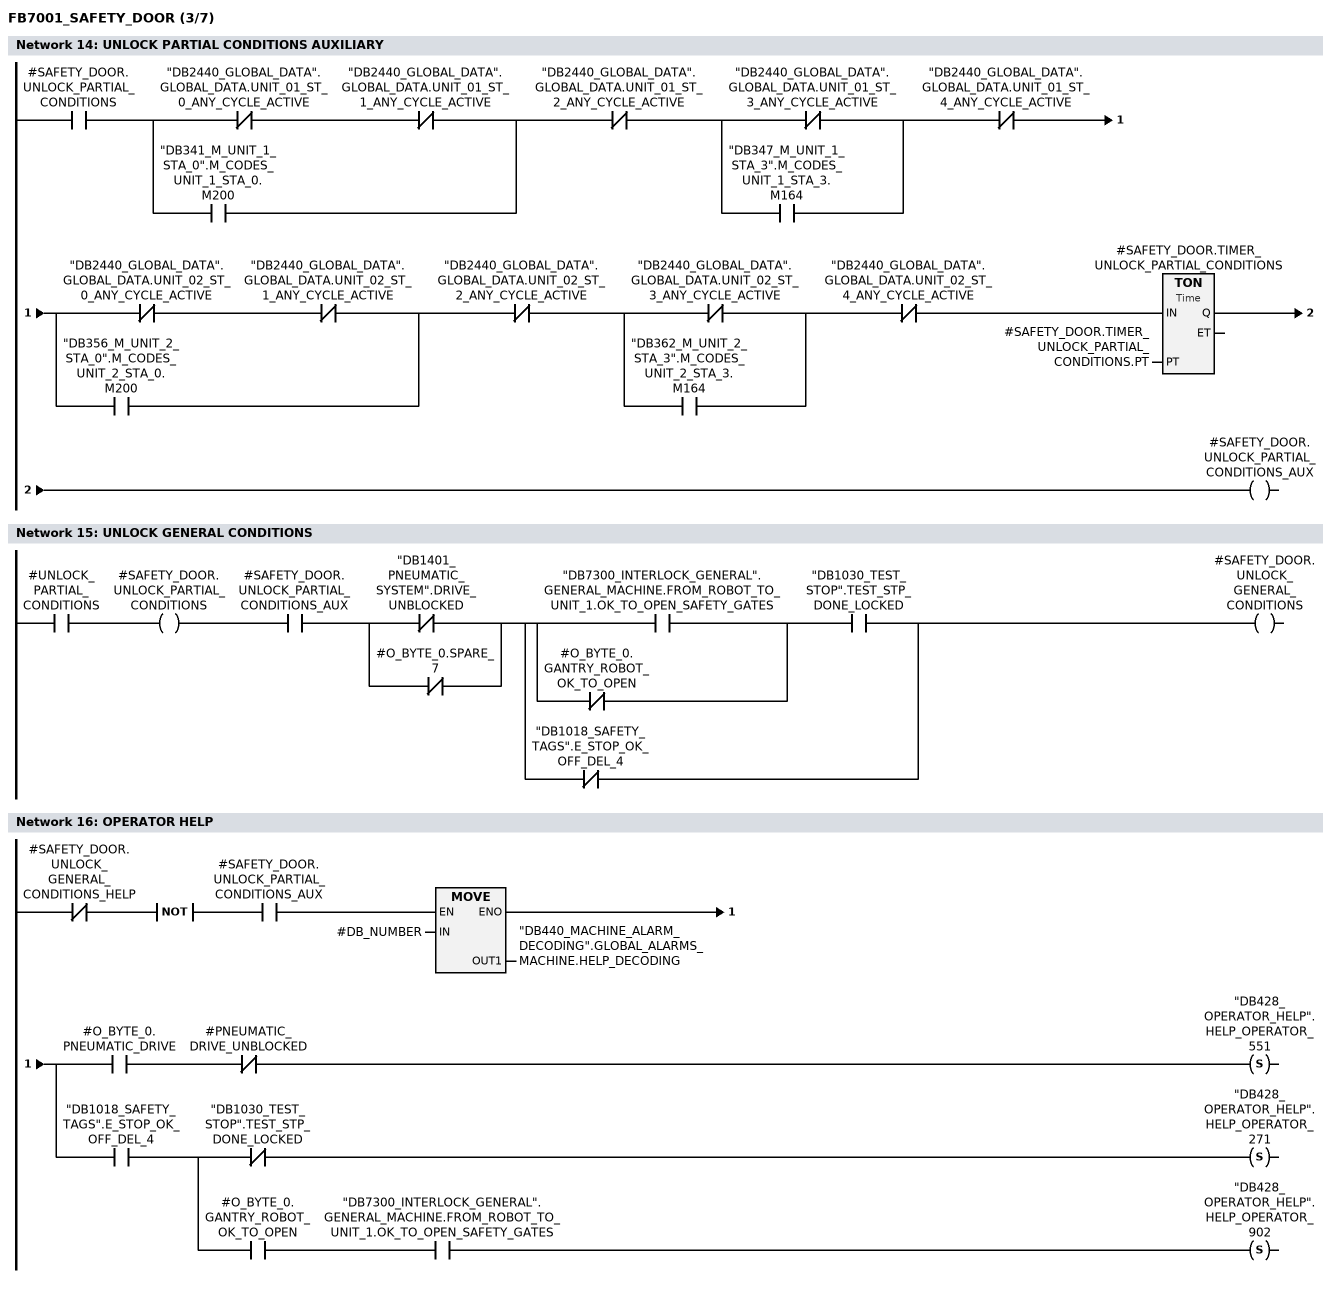
   RUNG wire#powerrail
      Contact( #SAFETY_DOOR.UNLOCK_PARTIAL_CONDITIONS )
      wire#w1
      I_Contact( "DB2440_GLOBAL_DATA".GLOBAL_DATA.UNIT_01_ST_0_ANY_CYCLE_ACTIVE )
      I_Contact( "DB2440_GLOBAL_DATA".GLOBAL_DATA.UNIT_01_ST_1_ANY_CYCLE_ACTIVE )
      wire#w2
      I_Contact( "DB2440_GLOBAL_DATA".GLOBAL_DATA.UNIT_01_ST_2_ANY_CYCLE_ACTIVE )
      wire#w3
      I_Contact( "DB2440_GLOBAL_DATA".GLOBAL_DATA.UNIT_01_ST_3_ANY_CYCLE_ACTIVE )
      wire#w4
      I_Contact( "DB2440_GLOBAL_DATA".GLOBAL_DATA.UNIT_01_ST_4_ANY_CYCLE_ACTIVE )
      wire#w5
      I_Contact( "DB2440_GLOBAL_DATA".GLOBAL_DATA.UNIT_02_ST_0_ANY_CYCLE_ACTIVE )
      I_Contact( "DB2440_GLOBAL_DATA".GLOBAL_DATA.UNIT_02_ST_1_ANY_CYCLE_ACTIVE )
      wire#w6
      I_Contact( "DB2440_GLOBAL_DATA".GLOBAL_DATA.UNIT_02_ST_2_ANY_CYCLE_ACTIVE )
      wire#w7
      I_Contact( "DB2440_GLOBAL_DATA".GLOBAL_DATA.UNIT_02_ST_3_ANY_CYCLE_ACTIVE )
      wire#w8
      I_Contact( "DB2440_GLOBAL_DATA".GLOBAL_DATA.UNIT_02_ST_4_ANY_CYCLE_ACTIVE )
      { S7_Templates := "time_type := Time" } #SAFETY_DOOR.TIMER_UNLOCK_PARTIAL_CONDITIONS.TON(pt := #SAFETY_DOOR.TIMER_UNLOCK_PARTIAL_CONDITIONS.PT, et =>)
      Coil( #SAFETY_DOOR.UNLOCK_PARTIAL_CONDITIONS_AUX )
   END_RUNG
   RUNG wire#w1
      Contact( "DB341_M_UNIT_1_STA_0".M_CODES_UNIT_1_STA_0.M200 )
   END_RUNG wire#w2
   RUNG wire#w3
      Contact( "DB347_M_UNIT_1_STA_3".M_CODES_UNIT_1_STA_3.M164 )
   END_RUNG wire#w4
   RUNG wire#w5
      Contact( "DB356_M_UNIT_2_STA_0".M_CODES_UNIT_2_STA_0.M200 )
   END_RUNG wire#w6
   RUNG wire#w7
      Contact( "DB362_M_UNIT_2_STA_3".M_CODES_UNIT_2_STA_3.M164 )
   END_RUNG wire#w8
   // the same network as SCL:
   #SAFETY_DOOR.TIMER_UNLOCK_PARTIAL_CONDITIONS.TON(IN := #SAFETY_DOOR.UNLOCK_PARTIAL_CONDITIONS AND ((NOT "DB2440_GLOBAL_DATA".GLOBAL_DATA.UNIT_01_ST_0_ANY_CYCLE_ACTIVE AND NOT "DB2440_GLOBAL_DATA".GLOBAL_DATA.UNIT_01_ST_1_ANY_CYCLE_ACTIVE) OR "DB341_M_UNIT_1_STA_0".M_CODES_UNIT_1_STA_0.M200) AND NOT "DB2440_GLOBAL_DATA".GLOBAL_DATA.UNIT_01_ST_2_ANY_CYCLE_ACTIVE AND (NOT "DB2440_GLOBAL_DATA".GLOBAL_DATA.UNIT_01_ST_3_ANY_CYCLE_ACTIVE OR "DB347_M_UNIT_1_STA_3".M_CODES_UNIT_1_STA_3.M164) AND NOT "DB2440_GLOBAL_DATA".GLOBAL_DATA.UNIT_01_ST_4_ANY_CYCLE_ACTIVE AND ((NOT "DB2440_GLOBAL_DATA".GLOBAL_DATA.UNIT_02_ST_0_ANY_CYCLE_ACTIVE AND NOT "DB2440_GLOBAL_DATA".GLOBAL_DATA.UNIT_02_ST_1_ANY_CYCLE_ACTIVE) OR "DB356_M_UNIT_2_STA_0".M_CODES_UNIT_2_STA_0.M200) AND NOT "DB2440_GLOBAL_DATA".GLOBAL_DATA.UNIT_02_ST_2_ANY_CYCLE_ACTIVE AND (NOT "DB2440_GLOBAL_DATA".GLOBAL_DATA.UNIT_02_ST_3_ANY_CYCLE_ACTIVE OR "DB362_M_UNIT_2_STA_3".M_CODES_UNIT_2_STA_3.M164) AND NOT "DB2440_GLOBAL_DATA".GLOBAL_DATA.UNIT_02_ST_4_ANY_CYCLE_ACTIVE,
                           PT := #SAFETY_DOOR.TIMER_UNLOCK_PARTIAL_CONDITIONS.PT);
   #SAFETY_DOOR.UNLOCK_PARTIAL_CONDITIONS_AUX := #SAFETY_DOOR.TIMER_UNLOCK_PARTIAL_CONDITIONS.Q;
END_REGION

REGION Network 15: UNLOCK GENERAL CONDITIONS
   RUNG wire#powerrail
      Contact( #UNLOCK_PARTIAL_CONDITIONS )
      Coil( #SAFETY_DOOR.UNLOCK_PARTIAL_CONDITIONS )
      Contact( #SAFETY_DOOR.UNLOCK_PARTIAL_CONDITIONS_AUX )
      wire#w1
      I_Contact( "DB1401_PNEUMATIC_SYSTEM".DRIVE_UNBLOCKED )
      wire#w2
      Contact( "DB7300_INTERLOCK_GENERAL".GENERAL_MACHINE.FROM_ROBOT_TO_UNIT_1.OK_TO_OPEN_SAFETY_GATES )
      wire#w3
      Contact( "DB1030_TEST_STOP".TEST_STP_DONE_LOCKED )
      wire#w4
      Coil( #SAFETY_DOOR.UNLOCK_GENERAL_CONDITIONS )
   END_RUNG
   RUNG wire#w1
      I_Contact( #O_BYTE_0.SPARE_7 )
   END_RUNG wire#w2
   RUNG wire#w2
      I_Contact( #O_BYTE_0.GANTRY_ROBOT_OK_TO_OPEN )
   END_RUNG wire#w3
   RUNG wire#w2
      I_Contact( "DB1018_SAFETY_TAGS".E_STOP_OK_OFF_DEL_4 )
   END_RUNG wire#w4
   // the same network as SCL:
   #SAFETY_DOOR.UNLOCK_PARTIAL_CONDITIONS := #UNLOCK_PARTIAL_CONDITIONS;
   #SAFETY_DOOR.UNLOCK_GENERAL_CONDITIONS := #UNLOCK_PARTIAL_CONDITIONS AND #SAFETY_DOOR.UNLOCK_PARTIAL_CONDITIONS_AUX AND (NOT "DB1401_PNEUMATIC_SYSTEM".DRIVE_UNBLOCKED OR NOT #O_BYTE_0.SPARE_7) AND ((("DB7300_INTERLOCK_GENERAL".GENERAL_MACHINE.FROM_ROBOT_TO_UNIT_1.OK_TO_OPEN_SAFETY_GATES OR NOT #O_BYTE_0.GANTRY_ROBOT_OK_TO_OPEN) AND "DB1030_TEST_STOP".TEST_STP_DONE_LOCKED) OR NOT "DB1018_SAFETY_TAGS".E_STOP_OK_OFF_DEL_4);
END_REGION

REGION Network 16: OPERATOR HELP
   RUNG wire#powerrail
      I_Contact( #SAFETY_DOOR.UNLOCK_GENERAL_CONDITIONS_HELP )
      Not()
      Contact( #SAFETY_DOOR.UNLOCK_PARTIAL_CONDITIONS_AUX )
      { S7_GenerateENO := "TRUE" } Move(in := #DB_NUMBER, out1 => "DB440_MACHINE_ALARM_DECODING".GLOBAL_ALARMS_MACHINE.HELP_DECODING)
      wire#w1
      Contact( #O_BYTE_0.PNEUMATIC_DRIVE )
      I_Contact( #PNEUMATIC_DRIVE_UNBLOCKED )
      S_Coil( "DB428_OPERATOR_HELP".HELP_OPERATOR_551 )
   END_RUNG
   RUNG wire#w1
      Contact( "DB1018_SAFETY_TAGS".E_STOP_OK_OFF_DEL_4 )
      wire#w2
      I_Contact( "DB1030_TEST_STOP".TEST_STP_DONE_LOCKED )
      S_Coil( "DB428_OPERATOR_HELP".HELP_OPERATOR_271 )
   END_RUNG
   RUNG wire#w2
      Contact( #O_BYTE_0.GANTRY_ROBOT_OK_TO_OPEN )
      Contact( "DB7300_INTERLOCK_GENERAL".GENERAL_MACHINE.FROM_ROBOT_TO_UNIT_1.OK_TO_OPEN_SAFETY_GATES )
      S_Coil( "DB428_OPERATOR_HELP".HELP_OPERATOR_902 )
   END_RUNG
   // the same network as SCL:
   // ENO of a box is taken as its EN; it also drops when the box reports an error
   #_w1 := NOT (NOT #SAFETY_DOOR.UNLOCK_GENERAL_CONDITIONS_HELP) AND #SAFETY_DOOR.UNLOCK_PARTIAL_CONDITIONS_AUX;
   IF #_w1 THEN "DB440_MACHINE_ALARM_DECODING".GLOBAL_ALARMS_MACHINE.HELP_DECODING := #DB_NUMBER; END_IF;
   IF #_w1 AND #O_BYTE_0.PNEUMATIC_DRIVE AND NOT #PNEUMATIC_DRIVE_UNBLOCKED THEN
       "DB428_OPERATOR_HELP".HELP_OPERATOR_551 := TRUE;
   END_IF;
   #_w2 := #_w1 AND "DB1018_SAFETY_TAGS".E_STOP_OK_OFF_DEL_4;
   IF #_w2 AND NOT "DB1030_TEST_STOP".TEST_STP_DONE_LOCKED THEN
       "DB428_OPERATOR_HELP".HELP_OPERATOR_271 := TRUE;
   END_IF;
   IF #_w2 AND #O_BYTE_0.GANTRY_ROBOT_OK_TO_OPEN AND "DB7300_INTERLOCK_GENERAL".GENERAL_MACHINE.FROM_ROBOT_TO_UNIT_1.OK_TO_OPEN_SAFETY_GATES THEN
       "DB428_OPERATOR_HELP".HELP_OPERATOR_902 := TRUE;
   END_IF;
END_REGION

REGION Network 17: UNLOCK MANUAL REQUEST
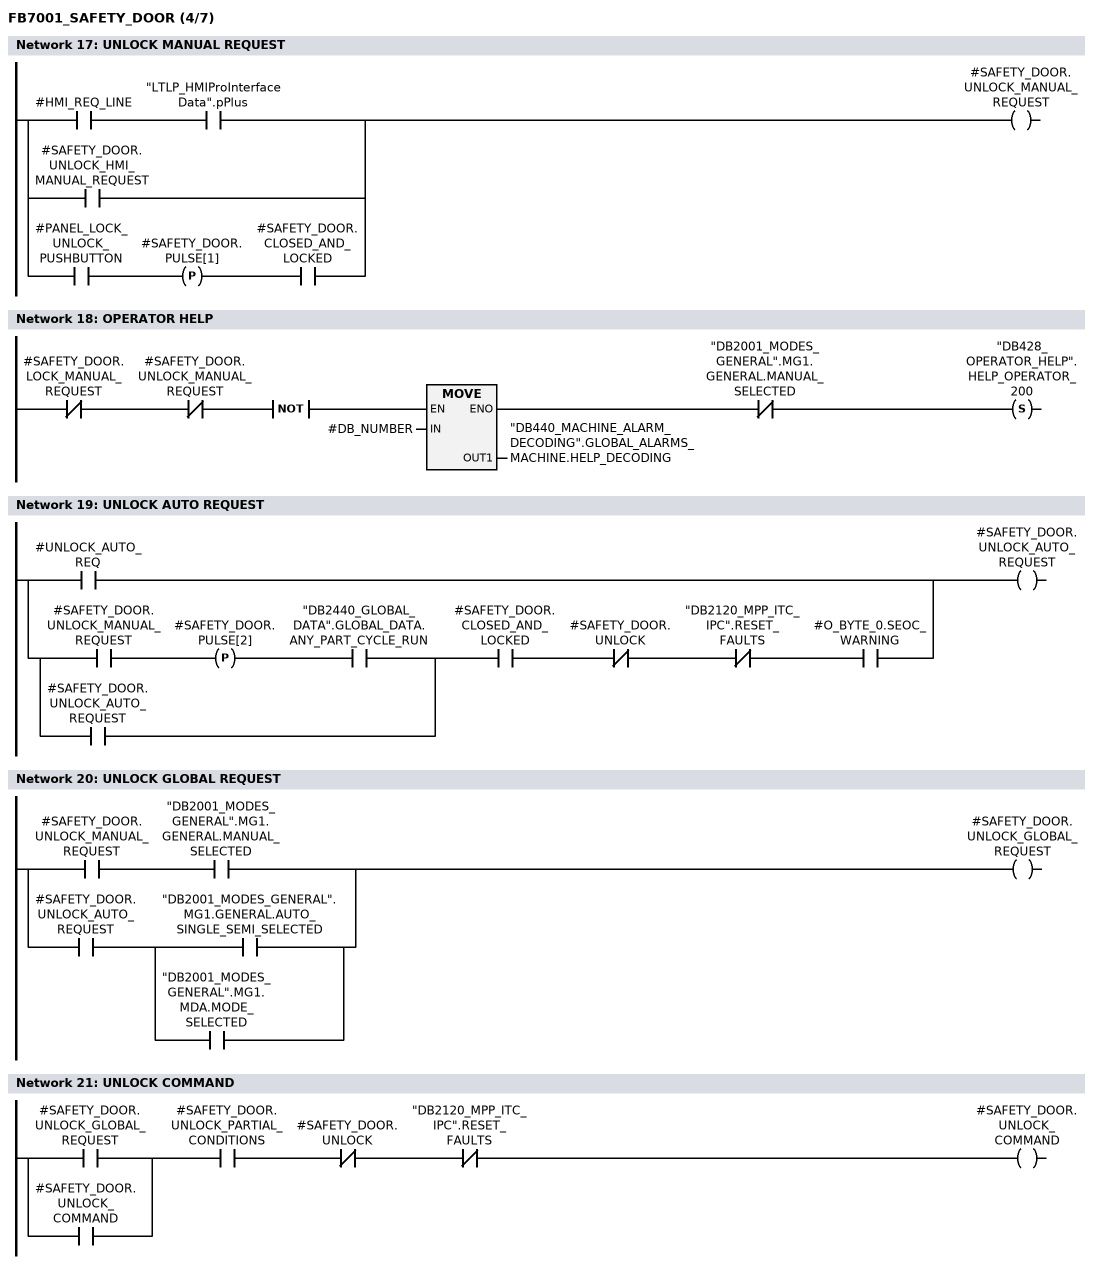
   RUNG wire#powerrail
      Contact( #HMI_REQ_LINE )
      Contact( "LTLP_HMIProInterfaceData".pPlus )
      wire#w1
      Coil( #SAFETY_DOOR.UNLOCK_MANUAL_REQUEST )
   END_RUNG
   RUNG wire#powerrail
      Contact( #SAFETY_DOOR.UNLOCK_HMI_MANUAL_REQUEST )
   END_RUNG wire#w1
   RUNG wire#powerrail
      Contact( #PANEL_LOCK_UNLOCK_PUSHBUTTON )
      P_Trig( #SAFETY_DOOR.PULSE[1] )
      Contact( #SAFETY_DOOR.CLOSED_AND_LOCKED )
   END_RUNG wire#w1
   // the same network as SCL:
   #_w1 := #PANEL_LOCK_UNLOCK_PUSHBUTTON AND NOT #SAFETY_DOOR.PULSE[1];   // rising edge
   #SAFETY_DOOR.PULSE[1] := #PANEL_LOCK_UNLOCK_PUSHBUTTON;
   #SAFETY_DOOR.UNLOCK_MANUAL_REQUEST := (#HMI_REQ_LINE AND "LTLP_HMIProInterfaceData".pPlus) OR #SAFETY_DOOR.UNLOCK_HMI_MANUAL_REQUEST OR (#_w1 AND #SAFETY_DOOR.CLOSED_AND_LOCKED);
END_REGION

REGION Network 18: OPERATOR HELP
   RUNG wire#powerrail
      I_Contact( #SAFETY_DOOR.LOCK_MANUAL_REQUEST )
      I_Contact( #SAFETY_DOOR.UNLOCK_MANUAL_REQUEST )
      Not()
      { S7_GenerateENO := "TRUE" } Move(in := #DB_NUMBER, out1 => "DB440_MACHINE_ALARM_DECODING".GLOBAL_ALARMS_MACHINE.HELP_DECODING)
      I_Contact( "DB2001_MODES_GENERAL".MG1.GENERAL.MANUAL_SELECTED )
      S_Coil( "DB428_OPERATOR_HELP".HELP_OPERATOR_200 )
   END_RUNG
   // the same network as SCL:
   // ENO of a box is taken as its EN; it also drops when the box reports an error
   #_w1 := NOT (NOT #SAFETY_DOOR.LOCK_MANUAL_REQUEST AND NOT #SAFETY_DOOR.UNLOCK_MANUAL_REQUEST);
   IF #_w1 THEN "DB440_MACHINE_ALARM_DECODING".GLOBAL_ALARMS_MACHINE.HELP_DECODING := #DB_NUMBER; END_IF;
   IF #_w1 AND NOT "DB2001_MODES_GENERAL".MG1.GENERAL.MANUAL_SELECTED THEN
       "DB428_OPERATOR_HELP".HELP_OPERATOR_200 := TRUE;
   END_IF;
END_REGION

REGION Network 19: UNLOCK AUTO REQUEST
   RUNG wire#powerrail
      Contact( #UNLOCK_AUTO_REQ )
      wire#w1
      Coil( #SAFETY_DOOR.UNLOCK_AUTO_REQUEST )
   END_RUNG
   RUNG wire#powerrail
      Contact( #SAFETY_DOOR.UNLOCK_MANUAL_REQUEST )
      P_Trig( #SAFETY_DOOR.PULSE[2] )
      Contact( "DB2440_GLOBAL_DATA".GLOBAL_DATA.ANY_PART_CYCLE_RUN )
      wire#w2
      Contact( #SAFETY_DOOR.CLOSED_AND_LOCKED )
      I_Contact( #SAFETY_DOOR.UNLOCK )
      I_Contact( "DB2120_MPP_ITC_IPC".RESET_FAULTS )
      Contact( #O_BYTE_0.SEOC_WARNING )
   END_RUNG wire#w1
   RUNG wire#powerrail
      Contact( #SAFETY_DOOR.UNLOCK_AUTO_REQUEST )
   END_RUNG wire#w2
   // the same network as SCL:
   #_w1 := #SAFETY_DOOR.UNLOCK_MANUAL_REQUEST AND NOT #SAFETY_DOOR.PULSE[2];   // rising edge
   #SAFETY_DOOR.PULSE[2] := #SAFETY_DOOR.UNLOCK_MANUAL_REQUEST;
   #SAFETY_DOOR.UNLOCK_AUTO_REQUEST := #UNLOCK_AUTO_REQ OR (((#_w1 AND "DB2440_GLOBAL_DATA".GLOBAL_DATA.ANY_PART_CYCLE_RUN) OR #SAFETY_DOOR.UNLOCK_AUTO_REQUEST) AND #SAFETY_DOOR.CLOSED_AND_LOCKED AND NOT #SAFETY_DOOR.UNLOCK AND NOT "DB2120_MPP_ITC_IPC".RESET_FAULTS AND #O_BYTE_0.SEOC_WARNING);
END_REGION

REGION Network 20: UNLOCK GLOBAL REQUEST
   RUNG wire#powerrail
      Contact( #SAFETY_DOOR.UNLOCK_MANUAL_REQUEST )
      Contact( "DB2001_MODES_GENERAL".MG1.GENERAL.MANUAL_SELECTED )
      wire#w1
      Coil( #SAFETY_DOOR.UNLOCK_GLOBAL_REQUEST )
   END_RUNG
   RUNG wire#powerrail
      Contact( #SAFETY_DOOR.UNLOCK_AUTO_REQUEST )
      wire#w2
      Contact( "DB2001_MODES_GENERAL".MG1.GENERAL.AUTO_SINGLE_SEMI_SELECTED )
   END_RUNG wire#w1
   RUNG wire#w2
      Contact( "DB2001_MODES_GENERAL".MG1.MDA.MODE_SELECTED )
   END_RUNG wire#w1
   // the same network as SCL:
   #SAFETY_DOOR.UNLOCK_GLOBAL_REQUEST := (#SAFETY_DOOR.UNLOCK_MANUAL_REQUEST AND "DB2001_MODES_GENERAL".MG1.GENERAL.MANUAL_SELECTED) OR (#SAFETY_DOOR.UNLOCK_AUTO_REQUEST AND ("DB2001_MODES_GENERAL".MG1.GENERAL.AUTO_SINGLE_SEMI_SELECTED OR "DB2001_MODES_GENERAL".MG1.MDA.MODE_SELECTED));
END_REGION

REGION Network 21: UNLOCK COMMAND
   RUNG wire#powerrail
      Contact( #SAFETY_DOOR.UNLOCK_GLOBAL_REQUEST )
      wire#w1
      Contact( #SAFETY_DOOR.UNLOCK_PARTIAL_CONDITIONS )
      I_Contact( #SAFETY_DOOR.UNLOCK )
      I_Contact( "DB2120_MPP_ITC_IPC".RESET_FAULTS )
      Coil( #SAFETY_DOOR.UNLOCK_COMMAND )
   END_RUNG
   RUNG wire#powerrail
      Contact( #SAFETY_DOOR.UNLOCK_COMMAND )
   END_RUNG wire#w1
   // the same network as SCL:
   #SAFETY_DOOR.UNLOCK_COMMAND := (#SAFETY_DOOR.UNLOCK_GLOBAL_REQUEST OR #SAFETY_DOOR.UNLOCK_COMMAND) AND #SAFETY_DOOR.UNLOCK_PARTIAL_CONDITIONS AND NOT #SAFETY_DOOR.UNLOCK AND NOT "DB2120_MPP_ITC_IPC".RESET_FAULTS;
END_REGION

REGION Network 22: UNLOCK
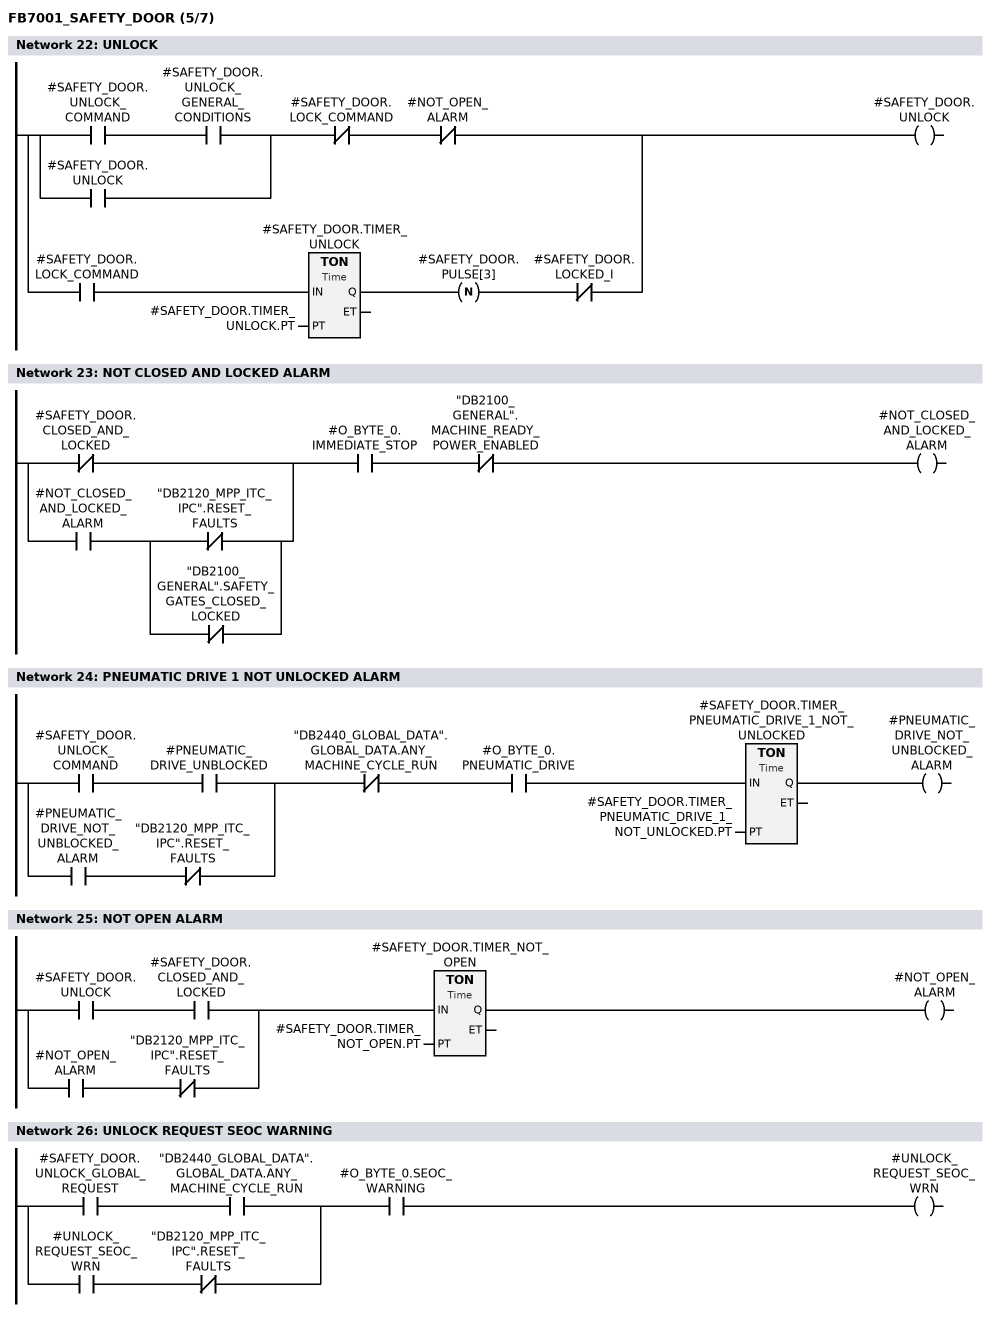
   RUNG wire#powerrail
      Contact( #SAFETY_DOOR.UNLOCK_COMMAND )
      Contact( #SAFETY_DOOR.UNLOCK_GENERAL_CONDITIONS )
      wire#w1
      I_Contact( #SAFETY_DOOR.LOCK_COMMAND )
      I_Contact( #NOT_OPEN_ALARM )
      wire#w2
      Coil( #SAFETY_DOOR.UNLOCK )
   END_RUNG
   RUNG wire#powerrail
      Contact( #SAFETY_DOOR.UNLOCK )
   END_RUNG wire#w1
   RUNG wire#powerrail
      Contact( #SAFETY_DOOR.LOCK_COMMAND )
      { S7_Templates := "time_type := Time" } #SAFETY_DOOR.TIMER_UNLOCK.TON(pt := #SAFETY_DOOR.TIMER_UNLOCK.PT, et =>)
      N_Trig( #SAFETY_DOOR.PULSE[3] )
      I_Contact( #SAFETY_DOOR.LOCKED_I )
   END_RUNG wire#w2
   // the same network as SCL:
   #SAFETY_DOOR.TIMER_UNLOCK.TON(IN := #SAFETY_DOOR.LOCK_COMMAND, PT := #SAFETY_DOOR.TIMER_UNLOCK.PT);
   #_w1 := NOT #SAFETY_DOOR.TIMER_UNLOCK.Q AND #SAFETY_DOOR.PULSE[3];   // falling edge
   #SAFETY_DOOR.PULSE[3] := #SAFETY_DOOR.TIMER_UNLOCK.Q;
   #SAFETY_DOOR.UNLOCK := (((#SAFETY_DOOR.UNLOCK_COMMAND AND #SAFETY_DOOR.UNLOCK_GENERAL_CONDITIONS) OR #SAFETY_DOOR.UNLOCK) AND NOT #SAFETY_DOOR.LOCK_COMMAND AND NOT #NOT_OPEN_ALARM) OR (#_w1 AND NOT #SAFETY_DOOR.LOCKED_I);
END_REGION

REGION Network 23: NOT CLOSED AND LOCKED ALARM
   RUNG wire#powerrail
      I_Contact( #SAFETY_DOOR.CLOSED_AND_LOCKED )
      wire#w1
      Contact( #O_BYTE_0.IMMEDIATE_STOP )
      I_Contact( "DB2100_GENERAL".MACHINE_READY_POWER_ENABLED )
      Coil( #NOT_CLOSED_AND_LOCKED_ALARM )
   END_RUNG
   RUNG wire#powerrail
      Contact( #NOT_CLOSED_AND_LOCKED_ALARM )
      wire#w2
      I_Contact( "DB2120_MPP_ITC_IPC".RESET_FAULTS )
   END_RUNG wire#w1
   RUNG wire#w2
      I_Contact( "DB2100_GENERAL".SAFETY_GATES_CLOSED_LOCKED )
   END_RUNG wire#w1
   // the same network as SCL:
   #NOT_CLOSED_AND_LOCKED_ALARM := (NOT #SAFETY_DOOR.CLOSED_AND_LOCKED OR (#NOT_CLOSED_AND_LOCKED_ALARM AND (NOT "DB2120_MPP_ITC_IPC".RESET_FAULTS OR NOT "DB2100_GENERAL".SAFETY_GATES_CLOSED_LOCKED))) AND #O_BYTE_0.IMMEDIATE_STOP AND NOT "DB2100_GENERAL".MACHINE_READY_POWER_ENABLED;
END_REGION

REGION Network 24: PNEUMATIC DRIVE 1 NOT UNLOCKED ALARM
   RUNG wire#powerrail
      Contact( #SAFETY_DOOR.UNLOCK_COMMAND )
      Contact( #PNEUMATIC_DRIVE_UNBLOCKED )
      wire#w1
      I_Contact( "DB2440_GLOBAL_DATA".GLOBAL_DATA.ANY_MACHINE_CYCLE_RUN )
      Contact( #O_BYTE_0.PNEUMATIC_DRIVE )
      { S7_Templates := "time_type := Time" } #SAFETY_DOOR.TIMER_PNEUMATIC_DRIVE_1_NOT_UNLOCKED.TON(pt := #SAFETY_DOOR.TIMER_PNEUMATIC_DRIVE_1_NOT_UNLOCKED.PT, et =>)
      Coil( #PNEUMATIC_DRIVE_NOT_UNBLOCKED_ALARM )
   END_RUNG
   RUNG wire#powerrail
      Contact( #PNEUMATIC_DRIVE_NOT_UNBLOCKED_ALARM )
      I_Contact( "DB2120_MPP_ITC_IPC".RESET_FAULTS )
   END_RUNG wire#w1
   // the same network as SCL:
   #SAFETY_DOOR.TIMER_PNEUMATIC_DRIVE_1_NOT_UNLOCKED.TON(IN := ((#SAFETY_DOOR.UNLOCK_COMMAND AND #PNEUMATIC_DRIVE_UNBLOCKED) OR (#PNEUMATIC_DRIVE_NOT_UNBLOCKED_ALARM AND NOT "DB2120_MPP_ITC_IPC".RESET_FAULTS)) AND NOT "DB2440_GLOBAL_DATA".GLOBAL_DATA.ANY_MACHINE_CYCLE_RUN AND #O_BYTE_0.PNEUMATIC_DRIVE,
                           PT := #SAFETY_DOOR.TIMER_PNEUMATIC_DRIVE_1_NOT_UNLOCKED.PT);
   #PNEUMATIC_DRIVE_NOT_UNBLOCKED_ALARM := #SAFETY_DOOR.TIMER_PNEUMATIC_DRIVE_1_NOT_UNLOCKED.Q;
END_REGION

REGION Network 25: NOT OPEN ALARM
   RUNG wire#powerrail
      Contact( #SAFETY_DOOR.UNLOCK )
      Contact( #SAFETY_DOOR.CLOSED_AND_LOCKED )
      wire#w1
      { S7_Templates := "time_type := Time" } #SAFETY_DOOR.TIMER_NOT_OPEN.TON(pt := #SAFETY_DOOR.TIMER_NOT_OPEN.PT, et =>)
      Coil( #NOT_OPEN_ALARM )
   END_RUNG
   RUNG wire#powerrail
      Contact( #NOT_OPEN_ALARM )
      I_Contact( "DB2120_MPP_ITC_IPC".RESET_FAULTS )
   END_RUNG wire#w1
   // the same network as SCL:
   #SAFETY_DOOR.TIMER_NOT_OPEN.TON(IN := (#SAFETY_DOOR.UNLOCK AND #SAFETY_DOOR.CLOSED_AND_LOCKED) OR (#NOT_OPEN_ALARM AND NOT "DB2120_MPP_ITC_IPC".RESET_FAULTS),
                           PT := #SAFETY_DOOR.TIMER_NOT_OPEN.PT);
   #NOT_OPEN_ALARM := #SAFETY_DOOR.TIMER_NOT_OPEN.Q;
END_REGION

REGION Network 26: UNLOCK REQUEST SEOC WARNING
   RUNG wire#powerrail
      Contact( #SAFETY_DOOR.UNLOCK_GLOBAL_REQUEST )
      Contact( "DB2440_GLOBAL_DATA".GLOBAL_DATA.ANY_MACHINE_CYCLE_RUN )
      wire#w1
      Contact( #O_BYTE_0.SEOC_WARNING )
      Coil( #UNLOCK_REQUEST_SEOC_WRN )
   END_RUNG
   RUNG wire#powerrail
      Contact( #UNLOCK_REQUEST_SEOC_WRN )
      I_Contact( "DB2120_MPP_ITC_IPC".RESET_FAULTS )
   END_RUNG wire#w1
   // the same network as SCL:
   #UNLOCK_REQUEST_SEOC_WRN := ((#SAFETY_DOOR.UNLOCK_GLOBAL_REQUEST AND "DB2440_GLOBAL_DATA".GLOBAL_DATA.ANY_MACHINE_CYCLE_RUN) OR (#UNLOCK_REQUEST_SEOC_WRN AND NOT "DB2120_MPP_ITC_IPC".RESET_FAULTS)) AND #O_BYTE_0.SEOC_WARNING;
END_REGION

REGION Network 27: IMMEDIATE STOP ALARMS
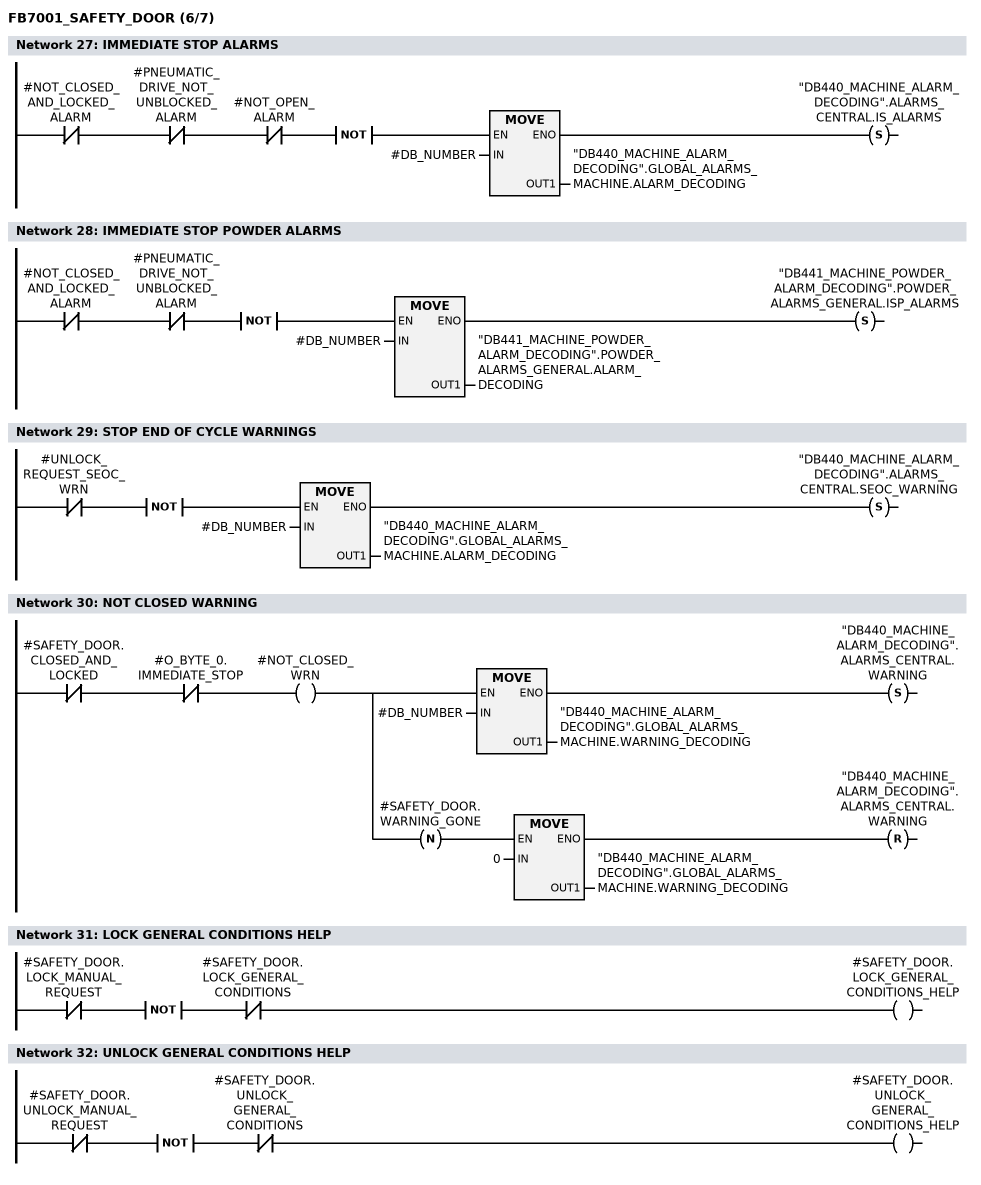
   RUNG wire#powerrail
      I_Contact( #NOT_CLOSED_AND_LOCKED_ALARM )
      I_Contact( #PNEUMATIC_DRIVE_NOT_UNBLOCKED_ALARM )
      I_Contact( #NOT_OPEN_ALARM )
      Not()
      { S7_GenerateENO := "TRUE" } Move(in := #DB_NUMBER, out1 => "DB440_MACHINE_ALARM_DECODING".GLOBAL_ALARMS_MACHINE.ALARM_DECODING)
      S_Coil( "DB440_MACHINE_ALARM_DECODING".ALARMS_CENTRAL.IS_ALARMS )
   END_RUNG
   // the same network as SCL:
   // ENO of a box is taken as its EN; it also drops when the box reports an error
   IF NOT (NOT #NOT_CLOSED_AND_LOCKED_ALARM AND NOT #PNEUMATIC_DRIVE_NOT_UNBLOCKED_ALARM AND NOT #NOT_OPEN_ALARM) THEN
       "DB440_MACHINE_ALARM_DECODING".GLOBAL_ALARMS_MACHINE.ALARM_DECODING := #DB_NUMBER;
       "DB440_MACHINE_ALARM_DECODING".ALARMS_CENTRAL.IS_ALARMS := TRUE;
   END_IF;
END_REGION

REGION Network 28: IMMEDIATE STOP POWDER ALARMS
   RUNG wire#powerrail
      I_Contact( #NOT_CLOSED_AND_LOCKED_ALARM )
      I_Contact( #PNEUMATIC_DRIVE_NOT_UNBLOCKED_ALARM )
      Not()
      { S7_GenerateENO := "TRUE" } Move(in := #DB_NUMBER, out1 => "DB441_MACHINE_POWDER_ALARM_DECODING".POWDER_ALARMS_GENERAL.ALARM_DECODING)
      S_Coil( "DB441_MACHINE_POWDER_ALARM_DECODING".POWDER_ALARMS_GENERAL.ISP_ALARMS )
   END_RUNG
   // the same network as SCL:
   // ENO of a box is taken as its EN; it also drops when the box reports an error
   IF NOT (NOT #NOT_CLOSED_AND_LOCKED_ALARM AND NOT #PNEUMATIC_DRIVE_NOT_UNBLOCKED_ALARM) THEN
       "DB441_MACHINE_POWDER_ALARM_DECODING".POWDER_ALARMS_GENERAL.ALARM_DECODING := #DB_NUMBER;
       "DB441_MACHINE_POWDER_ALARM_DECODING".POWDER_ALARMS_GENERAL.ISP_ALARMS := TRUE;
   END_IF;
END_REGION

REGION Network 29: STOP END OF CYCLE WARNINGS
   RUNG wire#powerrail
      I_Contact( #UNLOCK_REQUEST_SEOC_WRN )
      Not()
      { S7_GenerateENO := "TRUE" } Move(in := #DB_NUMBER, out1 => "DB440_MACHINE_ALARM_DECODING".GLOBAL_ALARMS_MACHINE.ALARM_DECODING)
      S_Coil( "DB440_MACHINE_ALARM_DECODING".ALARMS_CENTRAL.SEOC_WARNING )
   END_RUNG
   // the same network as SCL:
   // ENO of a box is taken as its EN; it also drops when the box reports an error
   IF NOT (NOT #UNLOCK_REQUEST_SEOC_WRN) THEN
       "DB440_MACHINE_ALARM_DECODING".GLOBAL_ALARMS_MACHINE.ALARM_DECODING := #DB_NUMBER;
       "DB440_MACHINE_ALARM_DECODING".ALARMS_CENTRAL.SEOC_WARNING := TRUE;
   END_IF;
END_REGION

REGION Network 30: NOT CLOSED WARNING
   RUNG wire#powerrail
      I_Contact( #SAFETY_DOOR.CLOSED_AND_LOCKED )
      I_Contact( #O_BYTE_0.IMMEDIATE_STOP )
      Coil( #NOT_CLOSED_WRN )
      wire#w1
      { S7_GenerateENO := "TRUE" } Move(in := #DB_NUMBER, out1 => "DB440_MACHINE_ALARM_DECODING".GLOBAL_ALARMS_MACHINE.WARNING_DECODING)
      S_Coil( "DB440_MACHINE_ALARM_DECODING".ALARMS_CENTRAL.WARNING )
   END_RUNG
   RUNG wire#w1
      N_Trig( #SAFETY_DOOR.WARNING_GONE )
      { S7_GenerateENO := "TRUE" } Move(in := 0, out1 => "DB440_MACHINE_ALARM_DECODING".GLOBAL_ALARMS_MACHINE.WARNING_DECODING)
      R_Coil( "DB440_MACHINE_ALARM_DECODING".ALARMS_CENTRAL.WARNING )
   END_RUNG
   // the same network as SCL:
   // ENO of a box is taken as its EN; it also drops when the box reports an error
   #NOT_CLOSED_WRN := NOT #SAFETY_DOOR.CLOSED_AND_LOCKED AND NOT #O_BYTE_0.IMMEDIATE_STOP;
   IF #NOT_CLOSED_WRN THEN
       "DB440_MACHINE_ALARM_DECODING".GLOBAL_ALARMS_MACHINE.WARNING_DECODING := #DB_NUMBER;
       "DB440_MACHINE_ALARM_DECODING".ALARMS_CENTRAL.WARNING := TRUE;
   END_IF;
   #_w1 := NOT #NOT_CLOSED_WRN AND #SAFETY_DOOR.WARNING_GONE;   // falling edge
   #SAFETY_DOOR.WARNING_GONE := #NOT_CLOSED_WRN;
   IF #_w1 THEN
       "DB440_MACHINE_ALARM_DECODING".GLOBAL_ALARMS_MACHINE.WARNING_DECODING := 0;
       "DB440_MACHINE_ALARM_DECODING".ALARMS_CENTRAL.WARNING := FALSE;
   END_IF;
END_REGION

REGION Network 31: LOCK GENERAL CONDITIONS HELP
   RUNG wire#powerrail
      I_Contact( #SAFETY_DOOR.LOCK_MANUAL_REQUEST )
      Not()
      I_Contact( #SAFETY_DOOR.LOCK_GENERAL_CONDITIONS )
      Coil( #SAFETY_DOOR.LOCK_GENERAL_CONDITIONS_HELP )
   END_RUNG
   // the same network as SCL:
   #SAFETY_DOOR.LOCK_GENERAL_CONDITIONS_HELP := NOT (NOT #SAFETY_DOOR.LOCK_MANUAL_REQUEST) AND NOT #SAFETY_DOOR.LOCK_GENERAL_CONDITIONS;
END_REGION

REGION Network 32: UNLOCK GENERAL CONDITIONS HELP
   RUNG wire#powerrail
      I_Contact( #SAFETY_DOOR.UNLOCK_MANUAL_REQUEST )
      Not()
      I_Contact( #SAFETY_DOOR.UNLOCK_GENERAL_CONDITIONS )
      Coil( #SAFETY_DOOR.UNLOCK_GENERAL_CONDITIONS_HELP )
   END_RUNG
   // the same network as SCL:
   #SAFETY_DOOR.UNLOCK_GENERAL_CONDITIONS_HELP := NOT (NOT #SAFETY_DOOR.UNLOCK_MANUAL_REQUEST) AND NOT #SAFETY_DOOR.UNLOCK_GENERAL_CONDITIONS;
END_REGION

REGION Network 33: HMI STATUS
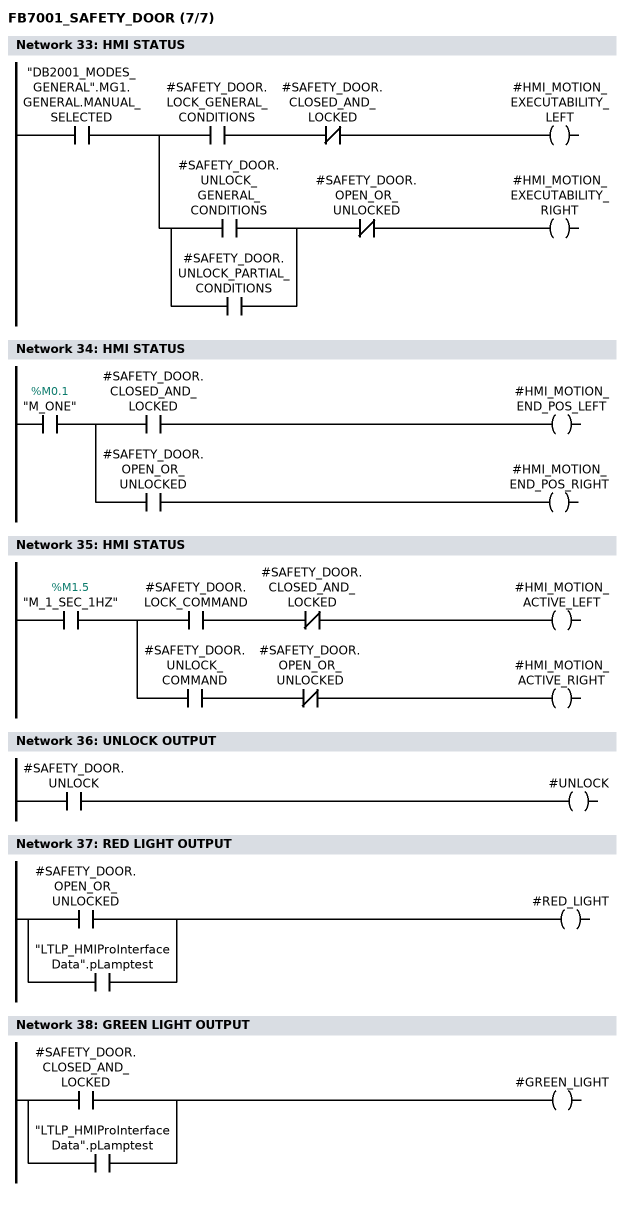
   RUNG wire#powerrail
      Contact( "DB2001_MODES_GENERAL".MG1.GENERAL.MANUAL_SELECTED )
      wire#w1
      Contact( #SAFETY_DOOR.LOCK_GENERAL_CONDITIONS )
      I_Contact( #SAFETY_DOOR.CLOSED_AND_LOCKED )
      Coil( #HMI_MOTION_EXECUTABILITY_LEFT )
   END_RUNG
   RUNG wire#w1
      Contact( #SAFETY_DOOR.UNLOCK_GENERAL_CONDITIONS )
      wire#w2
      I_Contact( #SAFETY_DOOR.OPEN_OR_UNLOCKED )
      Coil( #HMI_MOTION_EXECUTABILITY_RIGHT )
   END_RUNG
   RUNG wire#w1
      Contact( #SAFETY_DOOR.UNLOCK_PARTIAL_CONDITIONS )
   END_RUNG wire#w2
   // the same network as SCL:
   #HMI_MOTION_EXECUTABILITY_LEFT := "DB2001_MODES_GENERAL".MG1.GENERAL.MANUAL_SELECTED AND #SAFETY_DOOR.LOCK_GENERAL_CONDITIONS AND NOT #SAFETY_DOOR.CLOSED_AND_LOCKED;
   #HMI_MOTION_EXECUTABILITY_RIGHT := "DB2001_MODES_GENERAL".MG1.GENERAL.MANUAL_SELECTED AND (#SAFETY_DOOR.UNLOCK_GENERAL_CONDITIONS OR #SAFETY_DOOR.UNLOCK_PARTIAL_CONDITIONS) AND NOT #SAFETY_DOOR.OPEN_OR_UNLOCKED;
END_REGION

REGION Network 34: HMI STATUS
   RUNG wire#powerrail
      Contact( "M_ONE" )
      wire#w1
      Contact( #SAFETY_DOOR.CLOSED_AND_LOCKED )
      Coil( #HMI_MOTION_END_POS_LEFT )
   END_RUNG
   RUNG wire#w1
      Contact( #SAFETY_DOOR.OPEN_OR_UNLOCKED )
      Coil( #HMI_MOTION_END_POS_RIGHT )
   END_RUNG
   // the same network as SCL:
   #HMI_MOTION_END_POS_LEFT := "M_ONE" AND #SAFETY_DOOR.CLOSED_AND_LOCKED;
   #HMI_MOTION_END_POS_RIGHT := "M_ONE" AND #SAFETY_DOOR.OPEN_OR_UNLOCKED;
END_REGION

REGION Network 35: HMI STATUS
   RUNG wire#powerrail
      Contact( "M_1_SEC_1HZ" )
      wire#w1
      Contact( #SAFETY_DOOR.LOCK_COMMAND )
      I_Contact( #SAFETY_DOOR.CLOSED_AND_LOCKED )
      Coil( #HMI_MOTION_ACTIVE_LEFT )
   END_RUNG
   RUNG wire#w1
      Contact( #SAFETY_DOOR.UNLOCK_COMMAND )
      I_Contact( #SAFETY_DOOR.OPEN_OR_UNLOCKED )
      Coil( #HMI_MOTION_ACTIVE_RIGHT )
   END_RUNG
   // the same network as SCL:
   #HMI_MOTION_ACTIVE_LEFT := "M_1_SEC_1HZ" AND #SAFETY_DOOR.LOCK_COMMAND AND NOT #SAFETY_DOOR.CLOSED_AND_LOCKED;
   #HMI_MOTION_ACTIVE_RIGHT := "M_1_SEC_1HZ" AND #SAFETY_DOOR.UNLOCK_COMMAND AND NOT #SAFETY_DOOR.OPEN_OR_UNLOCKED;
END_REGION

REGION Network 36: UNLOCK OUTPUT
   RUNG wire#powerrail
      Contact( #SAFETY_DOOR.UNLOCK )
      Coil( #UNLOCK )
   END_RUNG
   // the same network as SCL:
   #UNLOCK := #SAFETY_DOOR.UNLOCK;
END_REGION

REGION Network 37: RED LIGHT OUTPUT
   RUNG wire#powerrail
      Contact( #SAFETY_DOOR.OPEN_OR_UNLOCKED )
      wire#w1
      Coil( #RED_LIGHT )
   END_RUNG
   RUNG wire#powerrail
      Contact( "LTLP_HMIProInterfaceData".pLamptest )
   END_RUNG wire#w1
   // the same network as SCL:
   #RED_LIGHT := #SAFETY_DOOR.OPEN_OR_UNLOCKED OR "LTLP_HMIProInterfaceData".pLamptest;
END_REGION

REGION Network 38: GREEN LIGHT OUTPUT
   RUNG wire#powerrail
      Contact( #SAFETY_DOOR.CLOSED_AND_LOCKED )
      wire#w1
      Coil( #GREEN_LIGHT )
   END_RUNG
   RUNG wire#powerrail
      Contact( "LTLP_HMIProInterfaceData".pLamptest )
   END_RUNG wire#w1
   // the same network as SCL:
   #GREEN_LIGHT := #SAFETY_DOOR.CLOSED_AND_LOCKED OR "LTLP_HMIProInterfaceData".pLamptest;
END_REGION
END_FUNCTION_BLOCK

FUNCTION "FC7200_HMI_FUNCTION" : Void   // FC7200, LAD
{ S7_Optimized_Access := 'FALSE' }
AUTHOR : ETXETAR
VERSION : 1.0
// stored: AutoNumber false, IsIECCheckEnabled false, SetENOAutomatically false, UDAEnableTagReadback false
   VAR_TEMP
      SCREEN_NAV : Bool;   // SCREEN NAVEGATION OPTION
      CNC_STATUS : Bool;   // CNC STATUS OPTION
      X : Int;
   END_VAR
   VAR CONSTANT
      TOTAL_SCREEN_NUM : Int := 89;
      FC_NUMBER : DInt := 7200;
   END_VAR
BEGIN

REGION Network 1: OPTIONS OFF
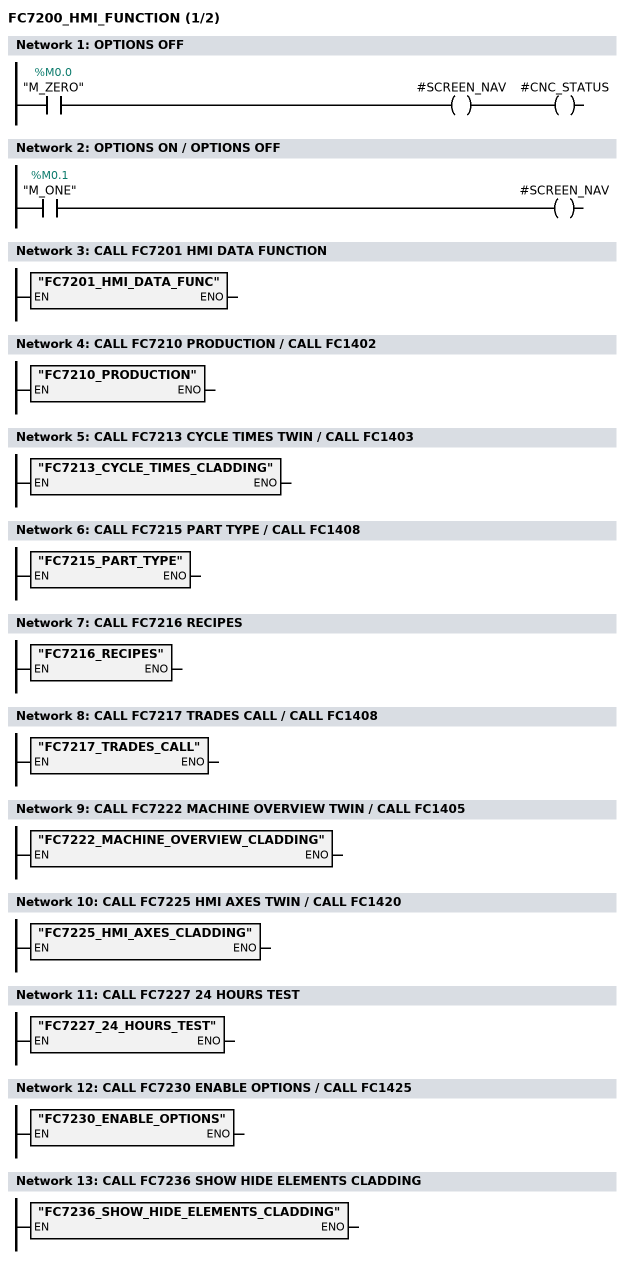
   RUNG wire#powerrail
      Contact( "M_ZERO" )
      Coil( #SCREEN_NAV )
      Coil( #CNC_STATUS )
   END_RUNG
   // the same network as SCL:
   #SCREEN_NAV := "M_ZERO";
   #CNC_STATUS := "M_ZERO";
END_REGION

REGION Network 2: OPTIONS ON / OPTIONS OFF
   RUNG wire#powerrail
      Contact( "M_ONE" )
      Coil( #SCREEN_NAV )
   END_RUNG
   // the same network as SCL:
   #SCREEN_NAV := "M_ONE";
END_REGION

REGION Network 3: CALL FC7201 HMI DATA FUNCTION
   RUNG wire#powerrail
      "FC7201_HMI_DATA_FUNC"()
   END_RUNG
   // the same network as SCL:
   "FC7201_HMI_DATA_FUNC"();
END_REGION

REGION Network 4: CALL FC7210 PRODUCTION / CALL FC1402
   RUNG wire#powerrail
      "FC7210_PRODUCTION"()
   END_RUNG
   // the same network as SCL:
   "FC7210_PRODUCTION"();
END_REGION

REGION Network 5: CALL FC7213 CYCLE TIMES TWIN / CALL FC1403
   RUNG wire#powerrail
      "FC7213_CYCLE_TIMES_CLADDING"()
   END_RUNG
   // the same network as SCL:
   "FC7213_CYCLE_TIMES_CLADDING"();
END_REGION

REGION Network 6: CALL FC7215 PART TYPE / CALL FC1408
   RUNG wire#powerrail
      "FC7215_PART_TYPE"()
   END_RUNG
   // the same network as SCL:
   "FC7215_PART_TYPE"();
END_REGION

REGION Network 7: CALL FC7216 RECIPES
   RUNG wire#powerrail
      "FC7216_RECIPES"()
   END_RUNG
   // the same network as SCL:
   "FC7216_RECIPES"();
END_REGION

REGION Network 8: CALL FC7217 TRADES CALL / CALL FC1408
   RUNG wire#powerrail
      "FC7217_TRADES_CALL"()
   END_RUNG
   // the same network as SCL:
   "FC7217_TRADES_CALL"();
END_REGION

REGION Network 9: CALL FC7222 MACHINE OVERVIEW TWIN / CALL FC1405
   RUNG wire#powerrail
      "FC7222_MACHINE_OVERVIEW_CLADDING"()
   END_RUNG
   // the same network as SCL:
   "FC7222_MACHINE_OVERVIEW_CLADDING"();
END_REGION

REGION Network 10: CALL FC7225 HMI AXES TWIN / CALL FC1420
   RUNG wire#powerrail
      "FC7225_HMI_AXES_CLADDING"()
   END_RUNG
   // the same network as SCL:
   "FC7225_HMI_AXES_CLADDING"();
END_REGION

REGION Network 11: CALL FC7227 24 HOURS TEST
   RUNG wire#powerrail
      "FC7227_24_HOURS_TEST"()
   END_RUNG
   // the same network as SCL:
   "FC7227_24_HOURS_TEST"();
END_REGION

REGION Network 12: CALL FC7230 ENABLE OPTIONS / CALL FC1425
   RUNG wire#powerrail
      "FC7230_ENABLE_OPTIONS"()
   END_RUNG
   // the same network as SCL:
   "FC7230_ENABLE_OPTIONS"();
END_REGION

REGION Network 13: CALL FC7236 SHOW HIDE ELEMENTS CLADDING
   RUNG wire#powerrail
      "FC7236_SHOW_HIDE_ELEMENTS_CLADDING"()
   END_RUNG
   // the same network as SCL:
   "FC7236_SHOW_HIDE_ELEMENTS_CLADDING"();
END_REGION

REGION Network 14: CALL FC7238 HMI WINCC OVERVIEW
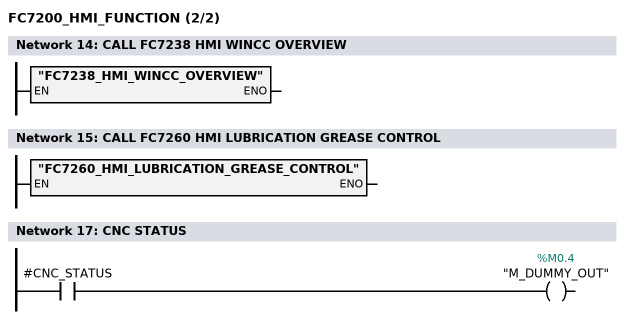
   RUNG wire#powerrail
      "FC7238_HMI_WINCC_OVERVIEW"()
   END_RUNG
   // the same network as SCL:
   "FC7238_HMI_WINCC_OVERVIEW"();
END_REGION

REGION Network 15: CALL FC7260 HMI LUBRICATION GREASE CONTROL
   RUNG wire#powerrail
      "FC7260_HMI_LUBRICATION_GREASE_CONTROL"()
   END_RUNG
   // the same network as SCL:
   "FC7260_HMI_LUBRICATION_GREASE_CONTROL"();
END_REGION

REGION Network 16 (SCL): SCREEN NAVIGATION

       IF #SCREEN_NAV THEN
           FOR #X := 11 TO #TOTAL_SCREEN_NUM DO
               IF "DB7200_HMI_FUNCTION".SCREEN_SELECTION[#X] THEN
                   "DB7200_HMI_FUNCTION".PLC_SCREEN_SELECTION :=INT_TO_WORD(#X);
               END_IF;
           END_FOR;
       END_IF;
END_REGION

REGION Network 17: CNC STATUS
   RUNG wire#powerrail
      Contact( #CNC_STATUS )
      Coil( "M_DUMMY_OUT" )
   END_RUNG
   // the same network as SCL:
   "M_DUMMY_OUT" := #CNC_STATUS;
END_REGION
END_FUNCTION

FUNCTION "FC8000_PART_STATUS" : Void   // FC8000, LAD
{ S7_Optimized_Access := 'FALSE' }
AUTHOR : ETXETAR
VERSION : 1.0
// BIT "PUN_A_PUN_B"
// 0 = THERE IS ONLY 1 "PUN DATA" OR "PART ID" 
// 1 = THERE ARE SEPARATE "PUN DATA" OR "PART ID" FOR PART A AND PART B
// 
// BIT "LIFTING_ONLY_1_POS"
// 0 = LIFTING HAS 2 OR 3 POSITIONS FOR AXIS W
// 1 = LIFTING HAS ONLY 1 POSITION FOR AXIS W
// stored: AutoNumber false, IsIECCheckEnabled false, SetENOAutomatically false, UDAEnableTagReadback false
   VAR_TEMP
      Workpiece_Screen : Int;
      Workpiece_Screen_selectd : Bool;
      zero : Byte;
      one : Byte;
      OPTION_ON : Bool;
      OPTION_OFF : Bool;
   END_VAR
BEGIN

REGION Network 1: OPTION OFF / OPTIONS OFF
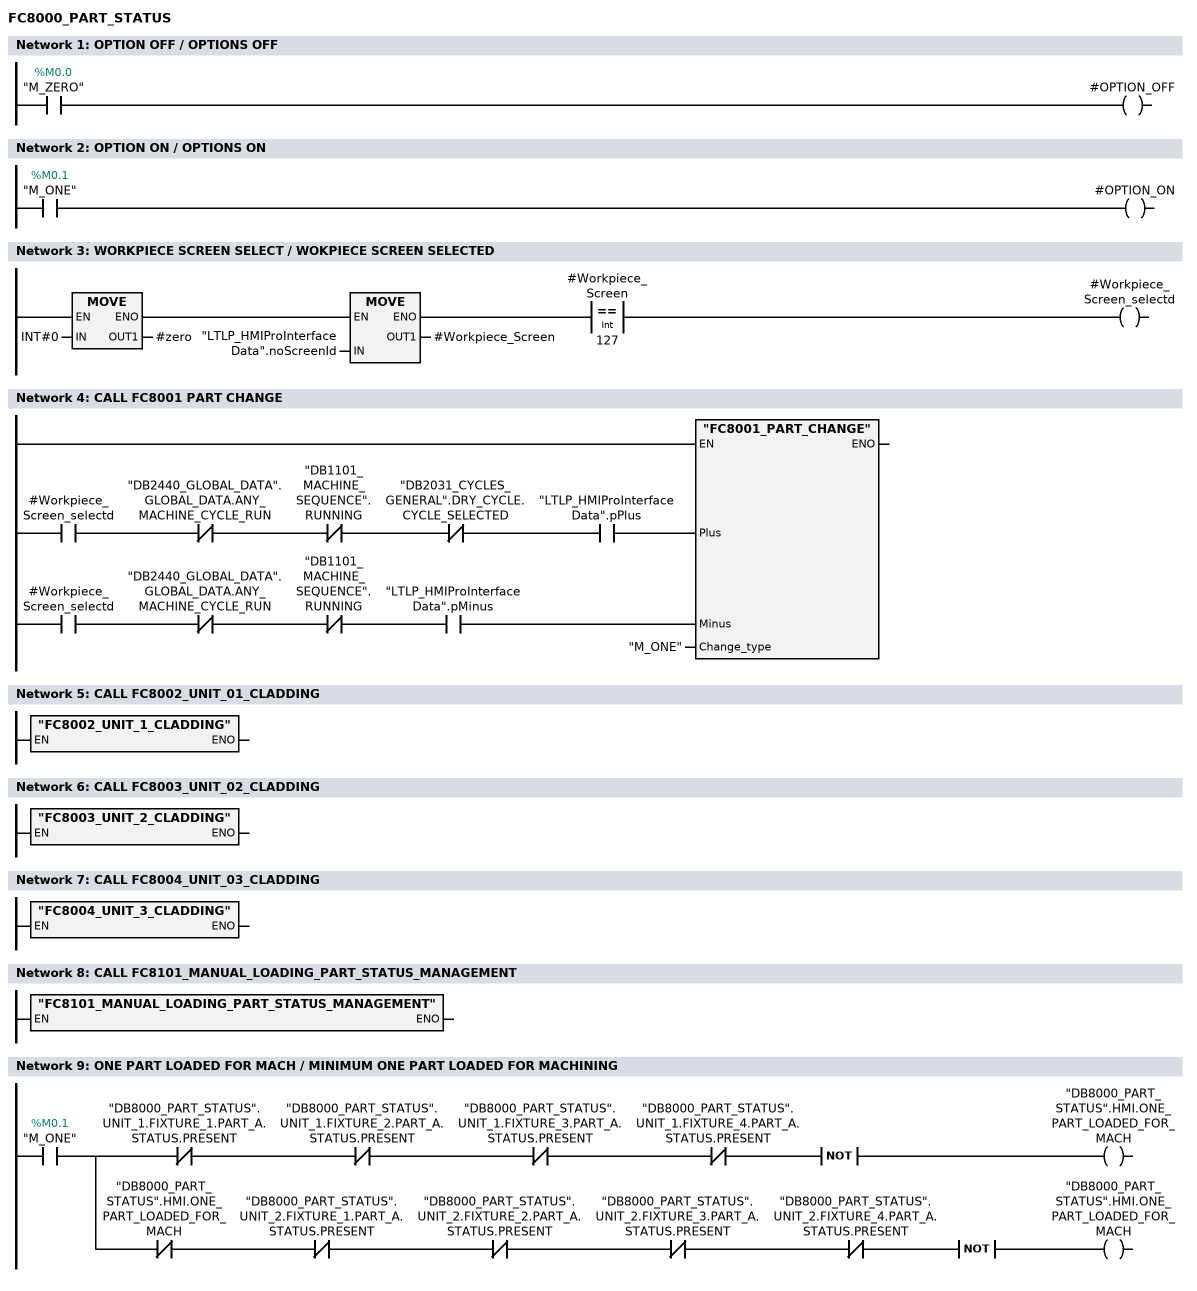
   RUNG wire#powerrail
      Contact( "M_ZERO" )
      Coil( #OPTION_OFF )
   END_RUNG
   // the same network as SCL:
   #OPTION_OFF := "M_ZERO";
END_REGION

REGION Network 2: OPTION ON / OPTIONS ON
   RUNG wire#powerrail
      Contact( "M_ONE" )
      Coil( #OPTION_ON )
   END_RUNG
   // the same network as SCL:
   #OPTION_ON := "M_ONE";
END_REGION

REGION Network 3: WORKPIECE SCREEN SELECT / WOKPIECE SCREEN SELECTED
   RUNG wire#powerrail
      { S7_GenerateENO := "TRUE" } Move(in := INT#0, out1 => #zero)
      { S7_GenerateENO := "TRUE" } Move(in := "LTLP_HMIProInterfaceData".noScreenId, out1 => #Workpiece_Screen)
      { S7_Templates := "SrcType := Int" } EQ_Contact(in1 := #Workpiece_Screen, in2 := 127)
      Coil( #Workpiece_Screen_selectd )
   END_RUNG
   // the same network as SCL:
   // ENO of a box is taken as its EN; it also drops when the box reports an error
   #zero := INT#0;
   #Workpiece_Screen := "LTLP_HMIProInterfaceData".noScreenId;
   #Workpiece_Screen_selectd := #Workpiece_Screen = 127;
END_REGION

REGION Network 4: CALL FC8001 PART CHANGE
   RUNG wire#powerrail
      "FC8001_PART_CHANGE"(Plus := wire#w1, Minus := wire#w2, Change_type := "M_ONE")
   END_RUNG
   RUNG wire#powerrail
      Contact( #Workpiece_Screen_selectd )
      I_Contact( "DB2440_GLOBAL_DATA".GLOBAL_DATA.ANY_MACHINE_CYCLE_RUN )
      I_Contact( "DB1101_MACHINE_SEQUENCE".RUNNING )
      I_Contact( "DB2031_CYCLES_GENERAL".DRY_CYCLE.CYCLE_SELECTED )
      Contact( "LTLP_HMIProInterfaceData".pPlus )
   END_RUNG wire#w1
   RUNG wire#powerrail
      Contact( #Workpiece_Screen_selectd )
      I_Contact( "DB2440_GLOBAL_DATA".GLOBAL_DATA.ANY_MACHINE_CYCLE_RUN )
      I_Contact( "DB1101_MACHINE_SEQUENCE".RUNNING )
      Contact( "LTLP_HMIProInterfaceData".pMinus )
   END_RUNG wire#w2
   // the same network as SCL:
   "FC8001_PART_CHANGE"(Plus := #Workpiece_Screen_selectd AND NOT "DB2440_GLOBAL_DATA".GLOBAL_DATA.ANY_MACHINE_CYCLE_RUN AND NOT "DB1101_MACHINE_SEQUENCE".RUNNING AND NOT "DB2031_CYCLES_GENERAL".DRY_CYCLE.CYCLE_SELECTED AND "LTLP_HMIProInterfaceData".pPlus,
                        Minus := #Workpiece_Screen_selectd AND NOT "DB2440_GLOBAL_DATA".GLOBAL_DATA.ANY_MACHINE_CYCLE_RUN AND NOT "DB1101_MACHINE_SEQUENCE".RUNNING AND "LTLP_HMIProInterfaceData".pMinus,
                        Change_type := "M_ONE");
END_REGION

REGION Network 5: CALL FC8002_UNIT_01_CLADDING
   RUNG wire#powerrail
      "FC8002_UNIT_1_CLADDING"()
   END_RUNG
   // the same network as SCL:
   "FC8002_UNIT_1_CLADDING"();
END_REGION

REGION Network 6: CALL FC8003_UNIT_02_CLADDING
   RUNG wire#powerrail
      "FC8003_UNIT_2_CLADDING"()
   END_RUNG
   // the same network as SCL:
   "FC8003_UNIT_2_CLADDING"();
END_REGION

REGION Network 7: CALL FC8004_UNIT_03_CLADDING
   RUNG wire#powerrail
      "FC8004_UNIT_3_CLADDING"()
   END_RUNG
   // the same network as SCL:
   "FC8004_UNIT_3_CLADDING"();
END_REGION

REGION Network 8: CALL FC8101_MANUAL_LOADING_PART_STATUS_MANAGEMENT
   RUNG wire#powerrail
      "FC8101_MANUAL_LOADING_PART_STATUS_MANAGEMENT"()
   END_RUNG
   // the same network as SCL:
   "FC8101_MANUAL_LOADING_PART_STATUS_MANAGEMENT"();
END_REGION

REGION Network 9: ONE PART LOADED FOR MACH / MINIMUM ONE PART LOADED FOR MACHINING
   RUNG wire#powerrail
      Contact( "M_ONE" )
      wire#w1
      I_Contact( "DB8000_PART_STATUS".UNIT_1.FIXTURE_1.PART_A.STATUS.PRESENT )
      I_Contact( "DB8000_PART_STATUS".UNIT_1.FIXTURE_2.PART_A.STATUS.PRESENT )
      I_Contact( "DB8000_PART_STATUS".UNIT_1.FIXTURE_3.PART_A.STATUS.PRESENT )
      I_Contact( "DB8000_PART_STATUS".UNIT_1.FIXTURE_4.PART_A.STATUS.PRESENT )
      Not()
      Coil( "DB8000_PART_STATUS".HMI.ONE_PART_LOADED_FOR_MACH )
   END_RUNG
   RUNG wire#w1
      I_Contact( "DB8000_PART_STATUS".HMI.ONE_PART_LOADED_FOR_MACH )
      I_Contact( "DB8000_PART_STATUS".UNIT_2.FIXTURE_1.PART_A.STATUS.PRESENT )
      I_Contact( "DB8000_PART_STATUS".UNIT_2.FIXTURE_2.PART_A.STATUS.PRESENT )
      I_Contact( "DB8000_PART_STATUS".UNIT_2.FIXTURE_3.PART_A.STATUS.PRESENT )
      I_Contact( "DB8000_PART_STATUS".UNIT_2.FIXTURE_4.PART_A.STATUS.PRESENT )
      Not()
      Coil( "DB8000_PART_STATUS".HMI.ONE_PART_LOADED_FOR_MACH )
   END_RUNG
   // the same network as SCL:
   "DB8000_PART_STATUS".HMI.ONE_PART_LOADED_FOR_MACH := NOT ("M_ONE" AND NOT "DB8000_PART_STATUS".UNIT_1.FIXTURE_1.PART_A.STATUS.PRESENT AND NOT "DB8000_PART_STATUS".UNIT_1.FIXTURE_2.PART_A.STATUS.PRESENT AND NOT "DB8000_PART_STATUS".UNIT_1.FIXTURE_3.PART_A.STATUS.PRESENT AND NOT "DB8000_PART_STATUS".UNIT_1.FIXTURE_4.PART_A.STATUS.PRESENT);
   "DB8000_PART_STATUS".HMI.ONE_PART_LOADED_FOR_MACH := NOT ("M_ONE" AND NOT "DB8000_PART_STATUS".HMI.ONE_PART_LOADED_FOR_MACH AND NOT "DB8000_PART_STATUS".UNIT_2.FIXTURE_1.PART_A.STATUS.PRESENT AND NOT "DB8000_PART_STATUS".UNIT_2.FIXTURE_2.PART_A.STATUS.PRESENT AND NOT "DB8000_PART_STATUS".UNIT_2.FIXTURE_3.PART_A.STATUS.PRESENT AND NOT "DB8000_PART_STATUS".UNIT_2.FIXTURE_4.PART_A.STATUS.PRESENT);
END_REGION
END_FUNCTION

FUNCTION "FC8001_PART_CHANGE" : Void   // FC8001, LAD
{ S7_Optimized_Access := 'FALSE' }
AUTHOR : ETXETAR
VERSION : 1.0
// Change the workpiece code (0x means decimal)
// => input identifier = 0x61 
// 
// When the workpiece code is changed to  317 (317 is entered in input field (5)) 
// on the 3rd station, the following will result:  
// 
// DB59.DBB80:input identifier = 0x61 
// DB59.DBB79: selected station = 0x03 
// DB59.DBW68: Code  = 317 (decimal) 
//  
// 
// Change workpiece status OK/NOK 
// => input ID 0x40, column ID 0x00
// 
// When the status of a workpiece F (= sixth workpiece) is changed at the 3rd 
// station, the following data contents apply:
// DB59.DBB80: Input ID 0x40 + workpiece no. 6 = 0x46
// DB59.DBB79: Selected station 3 = 0x03 
//  
// 
// Change workpiece status exists/does not exist 
// => input ID 0x40, column ID 0x40
// 
// When the status of a workpiece F (= sixth workpiece) is changed at the 3rd 
// station, the following data contents apply:
// DB59.DBB80: Input ID 0x40 + workpiece no. 6 = 0x46
// DB59.DBB79: Column code 0x40 + selected station 3 = 0x43
// stored: AutoNumber false, IsIECCheckEnabled false, SetENOAutomatically false, UDAEnableTagReadback false
   VAR_INPUT
      Plus : Bool;
      Minus : Bool;
      Change_type : Bool;
   END_VAR
   VAR_TEMP
      aux1 : Int;
      DBB79 : Int;
      DBB80 : Int;
      TypBCD : Word;
   END_VAR
BEGIN

NETWORK
TITLE = 
      L     "LTLP_HMIProInterfaceData".noFunctionLow;

      BTI;
      T     #DBB79;
      L     "LTLP_HMIProInterfaceData".noFunctionHigh;
      OPN   "LTLP_HMIProInterfaceData";
      BTI;
      T     #DBB80;

NETWORK
TITLE = Part type change request
      A     #Change_type;
      A(;
      L     #DBB80;
      L     61;
      ==I;
      );
      JCN   ok;
      L     #DBB79;  //Station number
      L     1;  //Station adress (1556,1560,1564)
      -I;
      L     4;
      *I;
      L     1556;
      +I;
      SLW   3;
      LAR1;  //Load pointer Program number
      L     "LTLP_HMIProInterfaceData".codeWorkpiece;  // Load part type decimal
      OPN   "LTLP_HMIProInterfaceData";
      ITB;  //Convert to BCD
      T     #TypBCD;  //Transfer to local
      L     #TypBCD.%B0;  //Load high byte
      T     DBB [AR1, P#0.0];  //Transfer to low byte
      L     #TypBCD.%B1;  //Load low byte
      T     DBB [AR1, P#1.0];  //Transfer to high byte

      L     #DBB79;  //Station number
      L     1;  //Station adress (1556,1560,1564)
      -I;
      L     2;
      *I;
      L     2822;
      +I;
      SLW   3;
      LAR1;
      L     "LTLP_HMIProInterfaceData".codeWorkpiece;
      OPN   "LTLP_HMIProInterfaceData";
      T     DBW [AR1, P#0.0];
      JU    fin1;

REGION Network 3
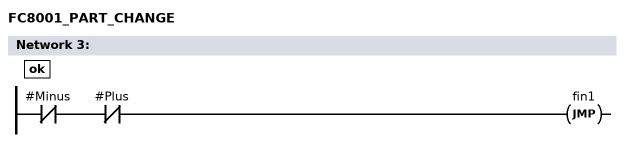
   Label( ok )
   RUNG wire#powerrail
      I_Contact( #Minus )
      I_Contact( #Plus )
      JumpCoil( fin1 )
   END_RUNG
   // the same network as SCL:
   ok:
   IF NOT #Minus AND NOT #Plus THEN GOTO fin1; END_IF;
END_REGION

NETWORK
TITLE = OK/Not OK change request

      L     #DBB79;
      L     40;
      >I;
      JC    pres;
      L     #DBB79;  //Station number
      L     1;  //Station adress (1556,1560,1564)
      -I;
      L     4;
      *I;
      L     1558;  //First OK adress
      +I;
      SLW   3;
      LAR1;  // load pointer

      L     #DBB80;  //part number (up to 8)
      L     40;
      -I;
      T     #aux1;
      L     4;  // if GT 4
      >I;
      JC    may;
      L     #aux1;  //Part number <=4
      L     2;
      *I;
      L     1;
      -I;
      TAR1;
      +I;
      LAR1;
      JU    cam1;
may:  L     1;  //part number >4
      SLW   3;
      +AR1;  //increase pointer 1 byte
      L     #aux1;
      L     2;
      *I;
      L     9;
      -I;
      TAR1;
      +I;
      LAR1;
cam1: A     #Minus;
      R     DBX [AR1, P#0.0];
      A     #Plus;
      S     DBX [AR1, P#0.0];
      JU    fin1;

NETWORK
TITLE = Part present change request

pres: L     #DBB79;
      L     40;
      >I;
      JCN   fin1;
      L     #DBB79;
      L     80;  //Up to 40 stations
      <=I;
      JCN   fin1;
      L     #DBB79;  //Station number
      L     41;  //Station adress (1556,1560,1564)
      -I;
      L     4;
      *I;
      L     1558;  //First OK adress
      +I;
      SLW   3;
      LAR1;  // load pointer

      L     #DBB80;  //part number (up to 8)
      L     40;
      -I;
      T     #aux1;
      L     4;  // if GT 4
      >I;
      JC    may1;
      L     #aux1;  //Part number <=4
      L     2;
      *I;
      L     2;
      -I;
      TAR1;
      +I;
      LAR1;
      JU    cam2;
may1: L     1;  //part number >4
      SLW   3;
      +AR1;  //increase pointer 1 byte
      L     #aux1;
      L     2;
      *I;
      L     10;
      -I;
      TAR1;
      +I;
      LAR1;
cam2: A     #Minus;
      R     DBX [AR1, P#0.0];
      A     #Plus;
      S     DBX [AR1, P#0.0];



NETWORK
TITLE = 
fin1: NOP   0;



END_FUNCTION

FUNCTION "FC10000_GENERAL" : Void   // FC10000, LAD
{ S7_Optimized_Access := 'TRUE' }
VERSION : 0.1
// stored: AutoNumber false, IsIECCheckEnabled false, SetENOAutomatically false, UDAEnableTagReadback false
BEGIN

REGION Network 1: CALL FC10200 PYROMETERS
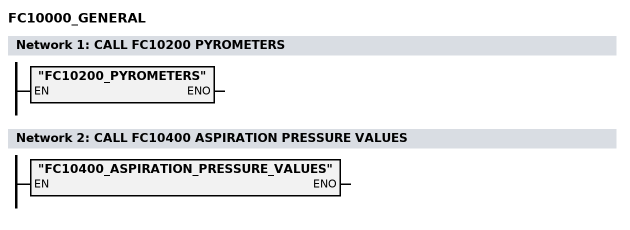
   RUNG wire#powerrail
      "FC10200_PYROMETERS"()
   END_RUNG
   // the same network as SCL:
   "FC10200_PYROMETERS"();
END_REGION

REGION Network 2: CALL FC10400 ASPIRATION PRESSURE VALUES
   RUNG wire#powerrail
      "FC10400_ASPIRATION_PRESSURE_VALUES"()
   END_RUNG
   // the same network as SCL:
   "FC10400_ASPIRATION_PRESSURE_VALUES"();
END_REGION
END_FUNCTION

FUNCTION "FC16000_OPC_UA_GENERAL" : Void   // FC16000, LAD
{ S7_Optimized_Access := 'TRUE' }
VERSION : 0.1
// stored: AutoNumber false, IsIECCheckEnabled false, SetENOAutomatically false, UDAEnableTagReadback false
BEGIN

REGION Network 1
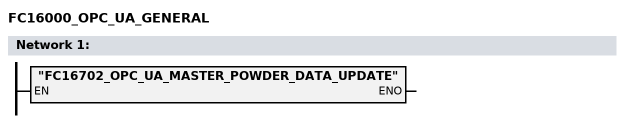
   RUNG wire#powerrail
      "FC16702_OPC_UA_MASTER_POWDER_DATA_UPDATE"()
   END_RUNG
   // the same network as SCL:
   "FC16702_OPC_UA_MASTER_POWDER_DATA_UPDATE"();
END_REGION
END_FUNCTION

ORGANIZATION_BLOCK "Cyclic interrupt"   // OB30, LAD, CyclicInterrupt
{ S7_Optimized_Access := 'TRUE' }
VERSION : 0.1
// stored: AutoNumber false, IsIECCheckEnabled false, SetENOAutomatically false
   VAR_INPUT
      Initial_Call : Bool;   // Initial call of this OB
      Event_Count : Int;   // Events discarded
   END_VAR
   VAR_TEMP
      LOOP_COUNT : Int;
   END_VAR
BEGIN

REGION Network 1: INITIALIZING OF ARRAY POINTERS FOR LOOP / Initializing of array pointers for loop
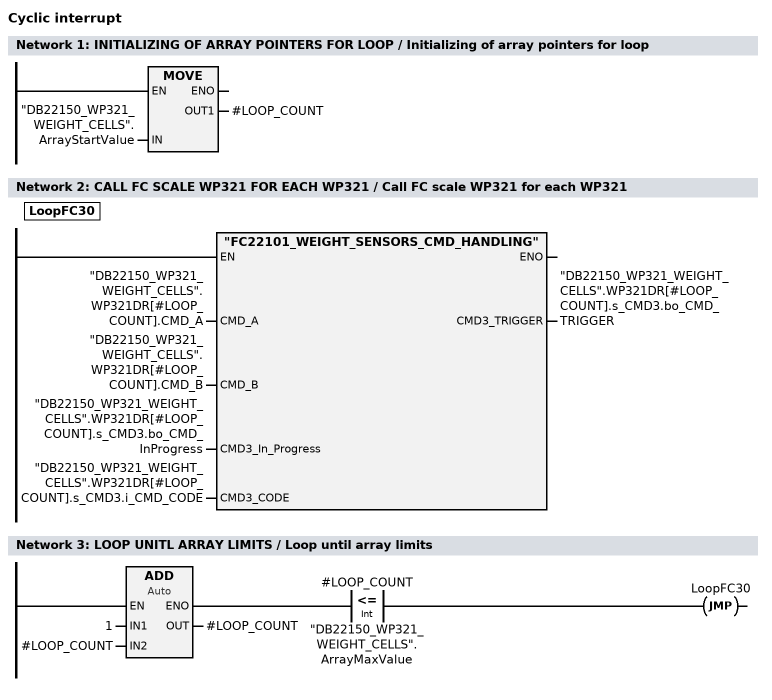
   RUNG wire#powerrail
      Move(in := "DB22150_WP321_WEIGHT_CELLS".ArrayStartValue, out1 => #LOOP_COUNT)
   END_RUNG
   // the same network as SCL:
   #LOOP_COUNT := "DB22150_WP321_WEIGHT_CELLS".ArrayStartValue;
END_REGION

REGION Network 2: CALL FC SCALE WP321 FOR EACH WP321 / Call FC scale WP321 for each WP321
   Label( LoopFC30 )
   RUNG wire#powerrail
      "FC22101_WEIGHT_SENSORS_CMD_HANDLING"(CMD_A := "DB22150_WP321_WEIGHT_CELLS".WP321DR[#LOOP_COUNT].CMD_A, CMD_B := "DB22150_WP321_WEIGHT_CELLS".WP321DR[#LOOP_COUNT].CMD_B, CMD3_In_Progress := "DB22150_WP321_WEIGHT_CELLS".WP321DR[#LOOP_COUNT].s_CMD3.bo_CMD_InProgress, CMD3_CODE := "DB22150_WP321_WEIGHT_CELLS".WP321DR[#LOOP_COUNT].s_CMD3.i_CMD_CODE, CMD3_TRIGGER => "DB22150_WP321_WEIGHT_CELLS".WP321DR[#LOOP_COUNT].s_CMD3.bo_CMD_TRIGGER)
   END_RUNG
   // the same network as SCL:
   LoopFC30:
   "FC22101_WEIGHT_SENSORS_CMD_HANDLING"(CMD_A := "DB22150_WP321_WEIGHT_CELLS".WP321DR[#LOOP_COUNT].CMD_A,
                           CMD_B := "DB22150_WP321_WEIGHT_CELLS".WP321DR[#LOOP_COUNT].CMD_B,
                           CMD3_In_Progress := "DB22150_WP321_WEIGHT_CELLS".WP321DR[#LOOP_COUNT].s_CMD3.bo_CMD_InProgress,
                           CMD3_CODE := "DB22150_WP321_WEIGHT_CELLS".WP321DR[#LOOP_COUNT].s_CMD3.i_CMD_CODE,
                           CMD3_TRIGGER => "DB22150_WP321_WEIGHT_CELLS".WP321DR[#LOOP_COUNT].s_CMD3.bo_CMD_TRIGGER);
END_REGION

REGION Network 3: LOOP UNITL ARRAY LIMITS / Loop until array limits
   RUNG wire#powerrail
      Add(in1 := 1, in2 := #LOOP_COUNT, out => #LOOP_COUNT)
      { S7_Templates := "SrcType := Int" } LE_Contact(in1 := #LOOP_COUNT, in2 := "DB22150_WP321_WEIGHT_CELLS".ArrayMaxValue)
      JumpCoil( LoopFC30 )
   END_RUNG
   // the same network as SCL:
   #LOOP_COUNT := 1 + #LOOP_COUNT;
   IF #LOOP_COUNT <= "DB22150_WP321_WEIGHT_CELLS".ArrayMaxValue THEN GOTO LoopFC30; END_IF;
END_REGION
END_ORGANIZATION_BLOCK

FUNCTION "FC22101_WEIGHT_SENSORS_CMD_HANDLING" : Void
{ S7_Optimized_Access := 'TRUE' }
VERSION : 0.1
   VAR_INPUT 
      CMD_A : Int;
      CMD_B : Int;
      CMD3_In_Progress : Bool;
   END_VAR

   VAR_OUTPUT 
      CMD3_TRIGGER : Bool;
   END_VAR

   VAR_IN_OUT 
      CMD3_CODE : Int;
   END_VAR


BEGIN
	IF (#CMD3_In_Progress=FALSE) THEN
	  IF (#CMD_A<>0) THEN
	    IF (#CMD_B<>0) THEN
	      IF (#CMD3_CODE=#CMD_A) THEN #CMD3_CODE:=#CMD_B;
	      ELSE #CMD3_CODE:=#CMD_A;
	      END_IF;
	    ELSE #CMD3_CODE:=#CMD_A;
	    END_IF;
	    #CMD3_TRIGGER:=TRUE;
	  ELSIF (#CMD_B<>0) THEN #CMD3_CODE:=#CMD_B; #CMD3_TRIGGER:=TRUE;
	  END_IF;
	 END_IF; 
END_FUNCTION

ORGANIZATION_BLOCK "OB100_RESTART"   // OB100, LAD, Startup
TITLE = "Complete Restart"
{ S7_Optimized_Access := 'FALSE' }
AUTHOR : ETXETAR
VERSION : 1.0
// stored: AutoNumber false, IsIECCheckEnabled false, SetENOAutomatically false
   VAR_TEMP
      OB100_EV_CLASS : Byte;
      OB100_STRTUP : Byte;
      OB100_PRIORITY : Byte;
      OB100_OB_NUMBR : Byte;
      OB100_RESERVED_1 : Byte;
      OB100_RESERVED_2 : Byte;
      OB100_STOP : Word;
      OB100_RESERVED_3 : Word;
      OB100_RESERVED_4 : Word;
      OB100_DATE_TIME : Date_And_Time;
      __PlcmigTempFillBits_20B0 : Array[0..7] of Bool;
   END_VAR
BEGIN

REGION Network 1: M_ONE / ESTABLISH "LOGIC 1" BIT
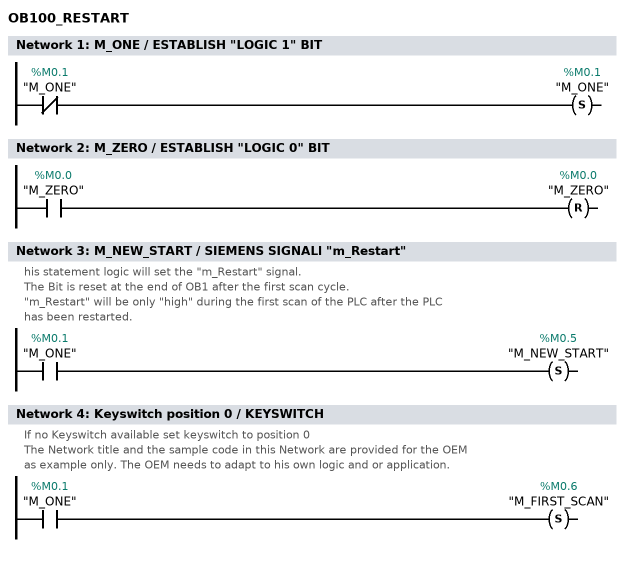
   RUNG wire#powerrail
      I_Contact( "M_ONE" )
      S_Coil( "M_ONE" )
   END_RUNG
   // the same network as SCL:
   IF NOT "M_ONE" THEN "M_ONE" := TRUE; END_IF;
END_REGION

REGION Network 2: M_ZERO / ESTABLISH "LOGIC 0" BIT
   RUNG wire#powerrail
      Contact( "M_ZERO" )
      R_Coil( "M_ZERO" )
   END_RUNG
   // the same network as SCL:
   IF "M_ZERO" THEN "M_ZERO" := FALSE; END_IF;
END_REGION

REGION Network 3: M_NEW_START / SIEMENS SIGNALl "m_Restart"
   // his statement logic will set the "m_Restart" signal.
   // The Bit is reset at the end of OB1 after the first scan cycle.
   // 
   // "m_Restart" will be only "high" during the first scan of the PLC after the PLC 
   // has been restarted.
   RUNG wire#powerrail
      Contact( "M_ONE" )
      S_Coil( "M_NEW_START" )
   END_RUNG
   // the same network as SCL:
   IF "M_ONE" THEN "M_NEW_START" := TRUE; END_IF;
END_REGION

REGION Network 4: Keyswitch position 0 / KEYSWITCH
   // If no Keyswitch available set keyswitch to position 0
   // 
   // The Network title and the sample code in this Network are provided for the OEM 
   // as example only. The OEM needs to adapt to his own logic and or application.
   RUNG wire#powerrail
      Contact( "M_ONE" )
      S_Coil( "M_FIRST_SCAN" )
   END_RUNG
   // the same network as SCL:
   IF "M_ONE" THEN "M_FIRST_SCAN" := TRUE; END_IF;
END_REGION
END_ORGANIZATION_BLOCK

ORGANIZATION_BLOCK "OB121_SYNCHRONF1"   // OB121, LAD, ProgrammingError
{ S7_Optimized_Access := 'FALSE' }
VERSION : 0.0
// stored: IsIECCheckEnabled false, SetENOAutomatically false
   VAR_TEMP
      TEMP0 : Byte;
      TEMP1 : Byte;
      TEMP2 : Byte;
      TEMP3 : Byte;
      TEMP4 : Byte;
      TEMP5 : Byte;
      TEMP6 : Word;
      TEMP7 : Word;
      TEMP8 : Word;
      TEMP9 : Date_And_Time;
   END_VAR
BEGIN
END_ORGANIZATION_BLOCK

ORGANIZATION_BLOCK "OB122_SYNCHRONF2"   // OB122, LAD, IOAccessError
{ S7_Optimized_Access := 'FALSE' }
VERSION : 0.0
// stored: IsIECCheckEnabled false, SetENOAutomatically false
   VAR_TEMP
      TEMP0 : Byte;
      TEMP1 : Byte;
      TEMP2 : Byte;
      TEMP3 : Byte;
      TEMP4 : Byte;
      TEMP5 : Byte;
      TEMP6 : Word;
      TEMP7 : Word;
      TEMP8 : Word;
      TEMP9 : Date_And_Time;
   END_VAR
BEGIN
END_ORGANIZATION_BLOCK

ORGANIZATION_BLOCK "OB40 Hardware interrupt"   // OB40, LAD, HardwareInterrupt
{ S7_Optimized_Access := 'TRUE' }
VERSION : 0.1
// stored: AutoNumber true, IsIECCheckEnabled false, SetENOAutomatically false
   VAR_INPUT
      LADDR : HW_IO;   // Hardware identifier
      USI : Word;   // User structure identifier
      IChannel : USInt;   // Interrupt channel number
      EventType : Byte;   // EventType
      PointAddr : DWord;
   END_VAR
   VAR_TEMP
      FLAG : Variant;
   END_VAR
BEGIN
END_ORGANIZATION_BLOCK

FUNCTION "FC15500_BDE" : Void   // FC15500, LAD
{ S7_Optimized_Access := 'TRUE' }
VERSION : 0.1
// stored: AutoNumber false, IsIECCheckEnabled false, SetENOAutomatically false, UDAEnableTagReadback false
BEGIN

REGION Network 1: FEED PART STATUS
   // PART_A/PART_B/PART_C/PART_D/PART_E
   // If the bit for the status of a feed part is to 0, the corresponding message text+ is available
   // is displayed in the image.
   // If the bit for the status of a feed part is set to 1, the corresponding message text + not available is displayed on the screen.
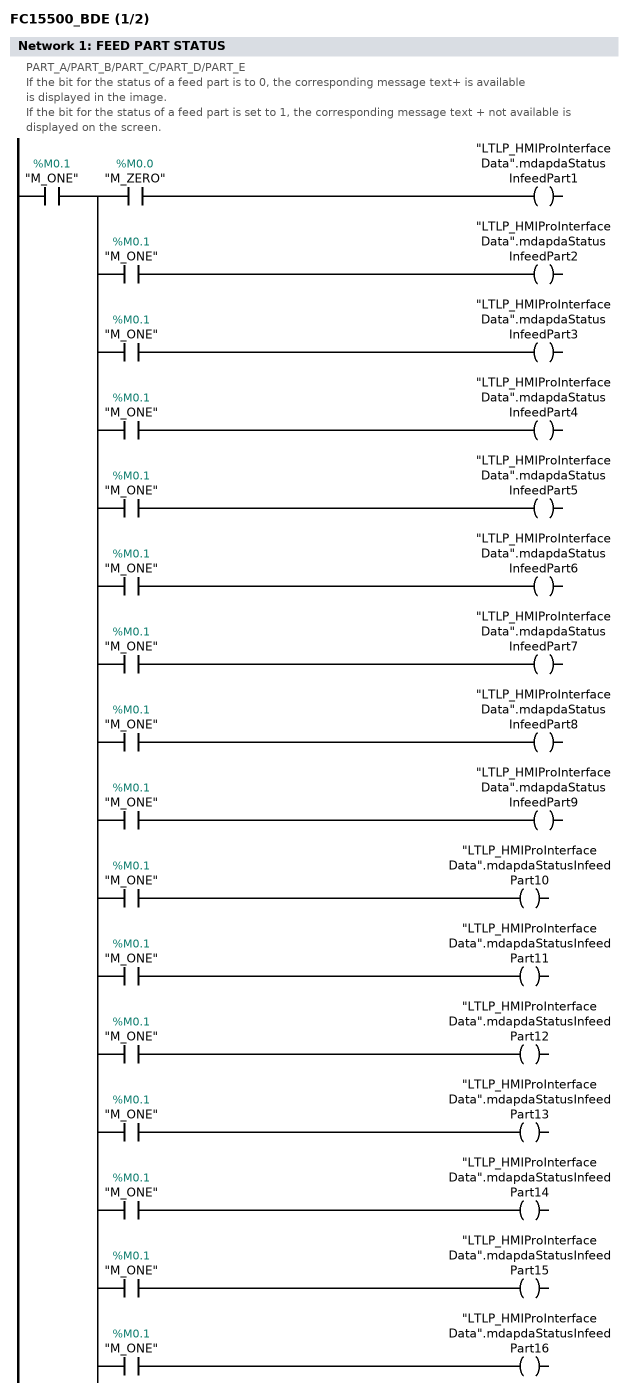
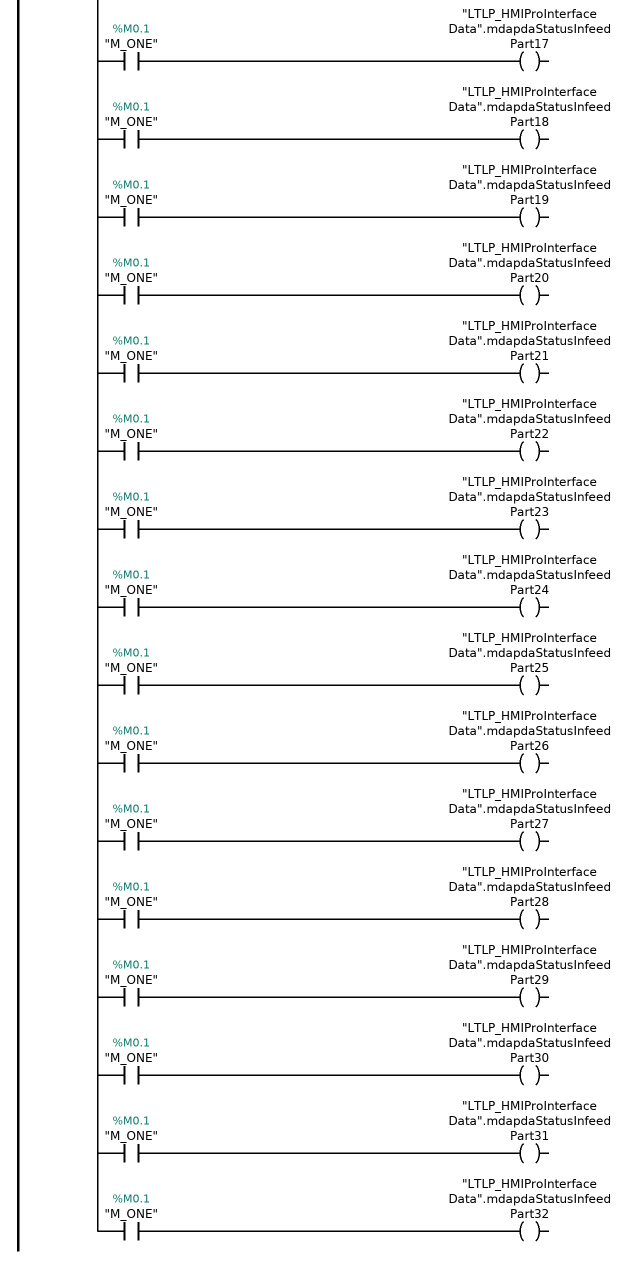
   RUNG wire#powerrail
      Contact( "M_ONE" )
      wire#w1
      Contact( "M_ZERO" )
      Coil( "LTLP_HMIProInterfaceData".mdapdaStatusInfeedPart1 )
   END_RUNG
   RUNG wire#w1
      Contact( "M_ONE" )
      Coil( "LTLP_HMIProInterfaceData".mdapdaStatusInfeedPart2 )
   END_RUNG
   RUNG wire#w1
      Contact( "M_ONE" )
      Coil( "LTLP_HMIProInterfaceData".mdapdaStatusInfeedPart3 )
   END_RUNG
   RUNG wire#w1
      Contact( "M_ONE" )
      Coil( "LTLP_HMIProInterfaceData".mdapdaStatusInfeedPart4 )
   END_RUNG
   RUNG wire#w1
      Contact( "M_ONE" )
      Coil( "LTLP_HMIProInterfaceData".mdapdaStatusInfeedPart5 )
   END_RUNG
   RUNG wire#w1
      Contact( "M_ONE" )
      Coil( "LTLP_HMIProInterfaceData".mdapdaStatusInfeedPart6 )
   END_RUNG
   RUNG wire#w1
      Contact( "M_ONE" )
      Coil( "LTLP_HMIProInterfaceData".mdapdaStatusInfeedPart7 )
   END_RUNG
   RUNG wire#w1
      Contact( "M_ONE" )
      Coil( "LTLP_HMIProInterfaceData".mdapdaStatusInfeedPart8 )
   END_RUNG
   RUNG wire#w1
      Contact( "M_ONE" )
      Coil( "LTLP_HMIProInterfaceData".mdapdaStatusInfeedPart9 )
   END_RUNG
   RUNG wire#w1
      Contact( "M_ONE" )
      Coil( "LTLP_HMIProInterfaceData".mdapdaStatusInfeedPart10 )
   END_RUNG
   RUNG wire#w1
      Contact( "M_ONE" )
      Coil( "LTLP_HMIProInterfaceData".mdapdaStatusInfeedPart11 )
   END_RUNG
   RUNG wire#w1
      Contact( "M_ONE" )
      Coil( "LTLP_HMIProInterfaceData".mdapdaStatusInfeedPart12 )
   END_RUNG
   RUNG wire#w1
      Contact( "M_ONE" )
      Coil( "LTLP_HMIProInterfaceData".mdapdaStatusInfeedPart13 )
   END_RUNG
   RUNG wire#w1
      Contact( "M_ONE" )
      Coil( "LTLP_HMIProInterfaceData".mdapdaStatusInfeedPart14 )
   END_RUNG
   RUNG wire#w1
      Contact( "M_ONE" )
      Coil( "LTLP_HMIProInterfaceData".mdapdaStatusInfeedPart15 )
   END_RUNG
   RUNG wire#w1
      Contact( "M_ONE" )
      Coil( "LTLP_HMIProInterfaceData".mdapdaStatusInfeedPart16 )
   END_RUNG
   RUNG wire#w1
      Contact( "M_ONE" )
      Coil( "LTLP_HMIProInterfaceData".mdapdaStatusInfeedPart17 )
   END_RUNG
   RUNG wire#w1
      Contact( "M_ONE" )
      Coil( "LTLP_HMIProInterfaceData".mdapdaStatusInfeedPart18 )
   END_RUNG
   RUNG wire#w1
      Contact( "M_ONE" )
      Coil( "LTLP_HMIProInterfaceData".mdapdaStatusInfeedPart19 )
   END_RUNG
   RUNG wire#w1
      Contact( "M_ONE" )
      Coil( "LTLP_HMIProInterfaceData".mdapdaStatusInfeedPart20 )
   END_RUNG
   RUNG wire#w1
      Contact( "M_ONE" )
      Coil( "LTLP_HMIProInterfaceData".mdapdaStatusInfeedPart21 )
   END_RUNG
   RUNG wire#w1
      Contact( "M_ONE" )
      Coil( "LTLP_HMIProInterfaceData".mdapdaStatusInfeedPart22 )
   END_RUNG
   RUNG wire#w1
      Contact( "M_ONE" )
      Coil( "LTLP_HMIProInterfaceData".mdapdaStatusInfeedPart23 )
   END_RUNG
   RUNG wire#w1
      Contact( "M_ONE" )
      Coil( "LTLP_HMIProInterfaceData".mdapdaStatusInfeedPart24 )
   END_RUNG
   RUNG wire#w1
      Contact( "M_ONE" )
      Coil( "LTLP_HMIProInterfaceData".mdapdaStatusInfeedPart25 )
   END_RUNG
   RUNG wire#w1
      Contact( "M_ONE" )
      Coil( "LTLP_HMIProInterfaceData".mdapdaStatusInfeedPart26 )
   END_RUNG
   RUNG wire#w1
      Contact( "M_ONE" )
      Coil( "LTLP_HMIProInterfaceData".mdapdaStatusInfeedPart27 )
   END_RUNG
   RUNG wire#w1
      Contact( "M_ONE" )
      Coil( "LTLP_HMIProInterfaceData".mdapdaStatusInfeedPart28 )
   END_RUNG
   RUNG wire#w1
      Contact( "M_ONE" )
      Coil( "LTLP_HMIProInterfaceData".mdapdaStatusInfeedPart29 )
   END_RUNG
   RUNG wire#w1
      Contact( "M_ONE" )
      Coil( "LTLP_HMIProInterfaceData".mdapdaStatusInfeedPart30 )
   END_RUNG
   RUNG wire#w1
      Contact( "M_ONE" )
      Coil( "LTLP_HMIProInterfaceData".mdapdaStatusInfeedPart31 )
   END_RUNG
   RUNG wire#w1
      Contact( "M_ONE" )
      Coil( "LTLP_HMIProInterfaceData".mdapdaStatusInfeedPart32 )
   END_RUNG
   // the same network as SCL:
   "LTLP_HMIProInterfaceData".mdapdaStatusInfeedPart1 := "M_ONE" AND "M_ZERO";
   "LTLP_HMIProInterfaceData".mdapdaStatusInfeedPart2 := "M_ONE" AND "M_ONE";
   "LTLP_HMIProInterfaceData".mdapdaStatusInfeedPart3 := "M_ONE" AND "M_ONE";
   "LTLP_HMIProInterfaceData".mdapdaStatusInfeedPart4 := "M_ONE" AND "M_ONE";
   "LTLP_HMIProInterfaceData".mdapdaStatusInfeedPart5 := "M_ONE" AND "M_ONE";
   "LTLP_HMIProInterfaceData".mdapdaStatusInfeedPart6 := "M_ONE" AND "M_ONE";
   "LTLP_HMIProInterfaceData".mdapdaStatusInfeedPart7 := "M_ONE" AND "M_ONE";
   "LTLP_HMIProInterfaceData".mdapdaStatusInfeedPart8 := "M_ONE" AND "M_ONE";
   "LTLP_HMIProInterfaceData".mdapdaStatusInfeedPart9 := "M_ONE" AND "M_ONE";
   "LTLP_HMIProInterfaceData".mdapdaStatusInfeedPart10 := "M_ONE" AND "M_ONE";
   "LTLP_HMIProInterfaceData".mdapdaStatusInfeedPart11 := "M_ONE" AND "M_ONE";
   "LTLP_HMIProInterfaceData".mdapdaStatusInfeedPart12 := "M_ONE" AND "M_ONE";
   "LTLP_HMIProInterfaceData".mdapdaStatusInfeedPart13 := "M_ONE" AND "M_ONE";
   "LTLP_HMIProInterfaceData".mdapdaStatusInfeedPart14 := "M_ONE" AND "M_ONE";
   "LTLP_HMIProInterfaceData".mdapdaStatusInfeedPart15 := "M_ONE" AND "M_ONE";
   "LTLP_HMIProInterfaceData".mdapdaStatusInfeedPart16 := "M_ONE" AND "M_ONE";
   "LTLP_HMIProInterfaceData".mdapdaStatusInfeedPart17 := "M_ONE" AND "M_ONE";
   "LTLP_HMIProInterfaceData".mdapdaStatusInfeedPart18 := "M_ONE" AND "M_ONE";
   "LTLP_HMIProInterfaceData".mdapdaStatusInfeedPart19 := "M_ONE" AND "M_ONE";
   "LTLP_HMIProInterfaceData".mdapdaStatusInfeedPart20 := "M_ONE" AND "M_ONE";
   "LTLP_HMIProInterfaceData".mdapdaStatusInfeedPart21 := "M_ONE" AND "M_ONE";
   "LTLP_HMIProInterfaceData".mdapdaStatusInfeedPart22 := "M_ONE" AND "M_ONE";
   "LTLP_HMIProInterfaceData".mdapdaStatusInfeedPart23 := "M_ONE" AND "M_ONE";
   "LTLP_HMIProInterfaceData".mdapdaStatusInfeedPart24 := "M_ONE" AND "M_ONE";
   "LTLP_HMIProInterfaceData".mdapdaStatusInfeedPart25 := "M_ONE" AND "M_ONE";
   "LTLP_HMIProInterfaceData".mdapdaStatusInfeedPart26 := "M_ONE" AND "M_ONE";
   "LTLP_HMIProInterfaceData".mdapdaStatusInfeedPart27 := "M_ONE" AND "M_ONE";
   "LTLP_HMIProInterfaceData".mdapdaStatusInfeedPart28 := "M_ONE" AND "M_ONE";
   "LTLP_HMIProInterfaceData".mdapdaStatusInfeedPart29 := "M_ONE" AND "M_ONE";
   "LTLP_HMIProInterfaceData".mdapdaStatusInfeedPart30 := "M_ONE" AND "M_ONE";
   "LTLP_HMIProInterfaceData".mdapdaStatusInfeedPart31 := "M_ONE" AND "M_ONE";
   "LTLP_HMIProInterfaceData".mdapdaStatusInfeedPart32 := "M_ONE" AND "M_ONE";
END_REGION

REGION Network 2: STATUS - SWITCHED ON/OFF
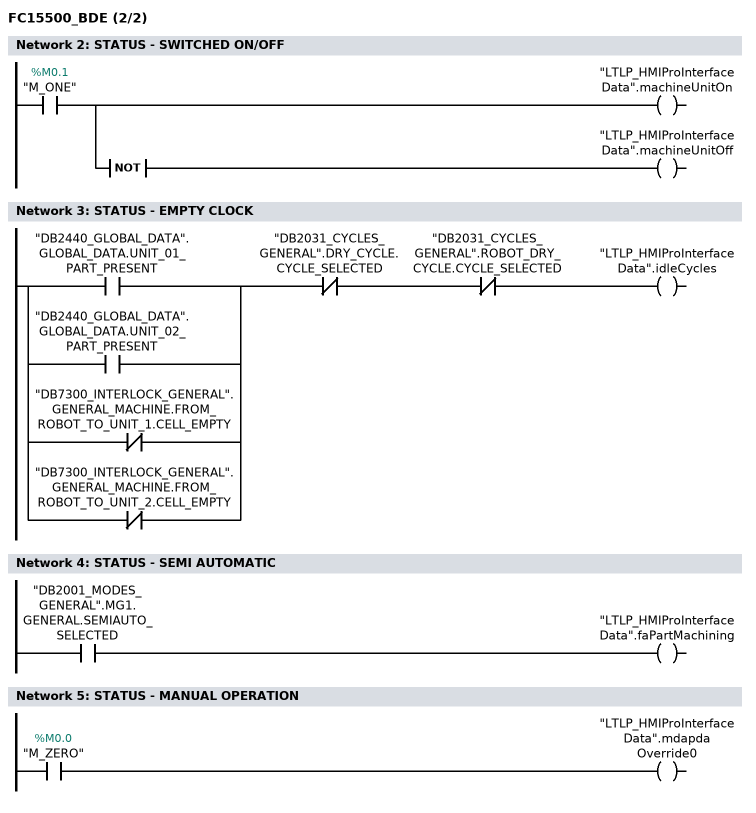
   RUNG wire#powerrail
      Contact( "M_ONE" )
      wire#w1
      Coil( "LTLP_HMIProInterfaceData".machineUnitOn )
   END_RUNG
   RUNG wire#w1
      Not()
      Coil( "LTLP_HMIProInterfaceData".machineUnitOff )
   END_RUNG
   // the same network as SCL:
   "LTLP_HMIProInterfaceData".machineUnitOn := "M_ONE";
   "LTLP_HMIProInterfaceData".machineUnitOff := NOT "M_ONE";
END_REGION

REGION Network 3: STATUS - EMPTY CLOCK
   RUNG wire#powerrail
      Contact( "DB2440_GLOBAL_DATA".GLOBAL_DATA.UNIT_01_PART_PRESENT )
      wire#w1
      I_Contact( "DB2031_CYCLES_GENERAL".DRY_CYCLE.CYCLE_SELECTED )
      I_Contact( "DB2031_CYCLES_GENERAL".ROBOT_DRY_CYCLE.CYCLE_SELECTED )
      Coil( "LTLP_HMIProInterfaceData".idleCycles )
   END_RUNG
   RUNG wire#powerrail
      Contact( "DB2440_GLOBAL_DATA".GLOBAL_DATA.UNIT_02_PART_PRESENT )
   END_RUNG wire#w1
   RUNG wire#powerrail
      I_Contact( "DB7300_INTERLOCK_GENERAL".GENERAL_MACHINE.FROM_ROBOT_TO_UNIT_1.CELL_EMPTY )
   END_RUNG wire#w1
   RUNG wire#powerrail
      I_Contact( "DB7300_INTERLOCK_GENERAL".GENERAL_MACHINE.FROM_ROBOT_TO_UNIT_2.CELL_EMPTY )
   END_RUNG wire#w1
   // the same network as SCL:
   "LTLP_HMIProInterfaceData".idleCycles := ("DB2440_GLOBAL_DATA".GLOBAL_DATA.UNIT_01_PART_PRESENT OR "DB2440_GLOBAL_DATA".GLOBAL_DATA.UNIT_02_PART_PRESENT OR NOT "DB7300_INTERLOCK_GENERAL".GENERAL_MACHINE.FROM_ROBOT_TO_UNIT_1.CELL_EMPTY OR NOT "DB7300_INTERLOCK_GENERAL".GENERAL_MACHINE.FROM_ROBOT_TO_UNIT_2.CELL_EMPTY) AND NOT "DB2031_CYCLES_GENERAL".DRY_CYCLE.CYCLE_SELECTED AND NOT "DB2031_CYCLES_GENERAL".ROBOT_DRY_CYCLE.CYCLE_SELECTED;
END_REGION

REGION Network 4: STATUS - SEMI AUTOMATIC
   RUNG wire#powerrail
      Contact( "DB2001_MODES_GENERAL".MG1.GENERAL.SEMIAUTO_SELECTED )
      Coil( "LTLP_HMIProInterfaceData".faPartMachining )
   END_RUNG
   // the same network as SCL:
   "LTLP_HMIProInterfaceData".faPartMachining := "DB2001_MODES_GENERAL".MG1.GENERAL.SEMIAUTO_SELECTED;
END_REGION

REGION Network 5: STATUS - MANUAL OPERATION
   RUNG wire#powerrail
      Contact( "M_ZERO" )
      Coil( "LTLP_HMIProInterfaceData".mdapdaOverride0 )
   END_RUNG
   // the same network as SCL:
   "LTLP_HMIProInterfaceData".mdapdaOverride0 := "M_ZERO";
END_REGION
END_FUNCTION

FUNCTION "FC2142_HOPPERS_SIGNAL_TOWER" : Void   // FC2142, LAD
{ S7_Optimized_Access := 'TRUE' }
VERSION : 0.1
// stored: AutoNumber false, IsIECCheckEnabled false, SetENOAutomatically false, UDAEnableTagReadback false
BEGIN

REGION Network 2: SIGNAL TOWER GREEN LIGHT OUTPUT / SIGNAL TOWER, GREEN LIGHT
   // M0.3 agregar las señales de starved y blocked de la celula / GREEN LIGHT
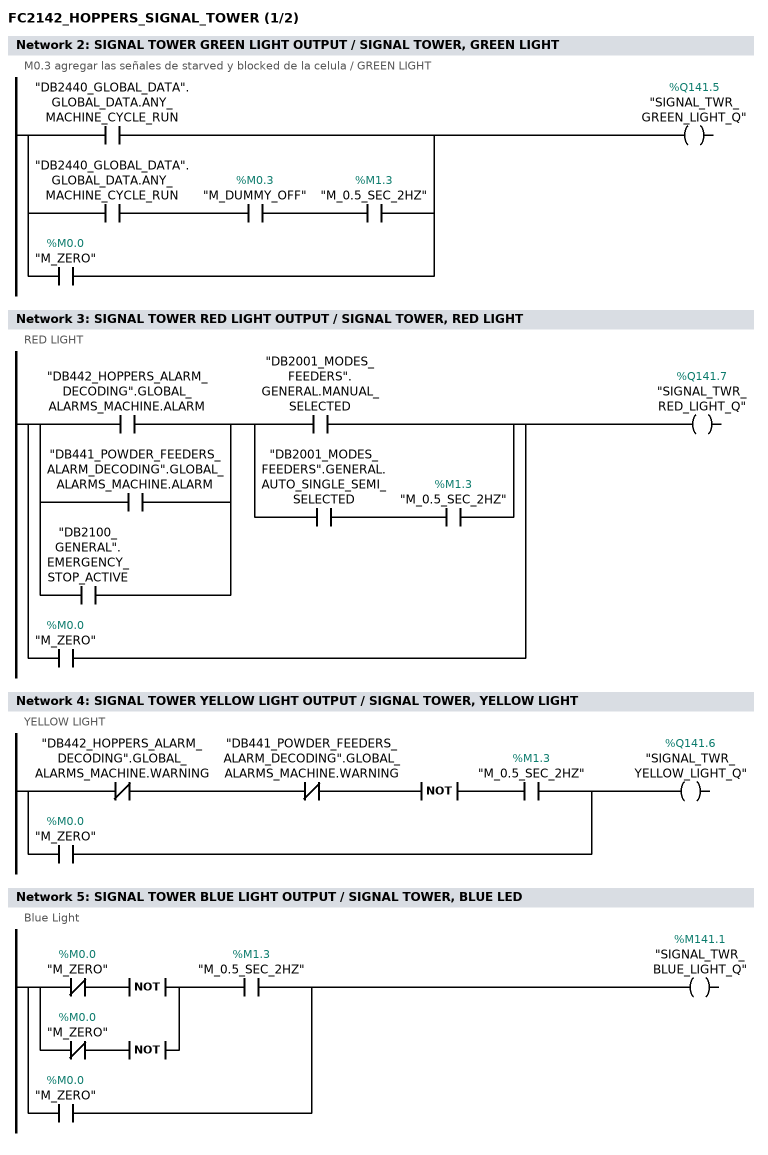
   RUNG wire#powerrail
      Contact( "DB2440_GLOBAL_DATA".GLOBAL_DATA.ANY_MACHINE_CYCLE_RUN )
      wire#w1
      Coil( "SIGNAL_TWR_GREEN_LIGHT_Q" )
   END_RUNG
   RUNG wire#powerrail
      Contact( "DB2440_GLOBAL_DATA".GLOBAL_DATA.ANY_MACHINE_CYCLE_RUN )
      Contact( "M_DUMMY_OFF" )
      Contact( "M_0.5_SEC_2HZ" )
   END_RUNG wire#w1
   RUNG wire#powerrail
      Contact( "M_ZERO" )
   END_RUNG wire#w1
   // the same network as SCL:
   "SIGNAL_TWR_GREEN_LIGHT_Q" := "DB2440_GLOBAL_DATA".GLOBAL_DATA.ANY_MACHINE_CYCLE_RUN OR ("DB2440_GLOBAL_DATA".GLOBAL_DATA.ANY_MACHINE_CYCLE_RUN AND "M_DUMMY_OFF" AND "M_0.5_SEC_2HZ") OR "M_ZERO";
END_REGION

REGION Network 3: SIGNAL TOWER RED LIGHT OUTPUT / SIGNAL TOWER, RED LIGHT
   // RED LIGHT
   RUNG wire#powerrail
      Contact( "DB442_HOPPERS_ALARM_DECODING".GLOBAL_ALARMS_MACHINE.ALARM )
      wire#w1
      Contact( "DB2001_MODES_FEEDERS".GENERAL.MANUAL_SELECTED )
      wire#w2
      Coil( "SIGNAL_TWR_RED_LIGHT_Q" )
   END_RUNG
   RUNG wire#powerrail
      Contact( "DB441_POWDER_FEEDERS_ALARM_DECODING".GLOBAL_ALARMS_MACHINE.ALARM )
   END_RUNG wire#w1
   RUNG wire#powerrail
      Contact( "DB2100_GENERAL".EMERGENCY_STOP_ACTIVE )
   END_RUNG wire#w1
   RUNG wire#w1
      Contact( "DB2001_MODES_FEEDERS".GENERAL.AUTO_SINGLE_SEMI_SELECTED )
      Contact( "M_0.5_SEC_2HZ" )
   END_RUNG wire#w2
   RUNG wire#powerrail
      Contact( "M_ZERO" )
   END_RUNG wire#w2
   // the same network as SCL:
   "SIGNAL_TWR_RED_LIGHT_Q" := (("DB442_HOPPERS_ALARM_DECODING".GLOBAL_ALARMS_MACHINE.ALARM OR "DB441_POWDER_FEEDERS_ALARM_DECODING".GLOBAL_ALARMS_MACHINE.ALARM OR "DB2100_GENERAL".EMERGENCY_STOP_ACTIVE) AND ("DB2001_MODES_FEEDERS".GENERAL.MANUAL_SELECTED OR ("DB2001_MODES_FEEDERS".GENERAL.AUTO_SINGLE_SEMI_SELECTED AND "M_0.5_SEC_2HZ"))) OR "M_ZERO";
END_REGION

REGION Network 4: SIGNAL TOWER YELLOW LIGHT OUTPUT / SIGNAL TOWER, YELLOW LIGHT
   // YELLOW LIGHT
   RUNG wire#powerrail
      I_Contact( "DB442_HOPPERS_ALARM_DECODING".GLOBAL_ALARMS_MACHINE.WARNING )
      I_Contact( "DB441_POWDER_FEEDERS_ALARM_DECODING".GLOBAL_ALARMS_MACHINE.WARNING )
      Not()
      Contact( "M_0.5_SEC_2HZ" )
      wire#w1
      Coil( "SIGNAL_TWR_YELLOW_LIGHT_Q" )
   END_RUNG
   RUNG wire#powerrail
      Contact( "M_ZERO" )
   END_RUNG wire#w1
   // the same network as SCL:
   "SIGNAL_TWR_YELLOW_LIGHT_Q" := (NOT (NOT "DB442_HOPPERS_ALARM_DECODING".GLOBAL_ALARMS_MACHINE.WARNING AND NOT "DB441_POWDER_FEEDERS_ALARM_DECODING".GLOBAL_ALARMS_MACHINE.WARNING) AND "M_0.5_SEC_2HZ") OR "M_ZERO";
END_REGION

REGION Network 5: SIGNAL TOWER BLUE LIGHT OUTPUT / SIGNAL TOWER, BLUE LED
   // Blue Light
   RUNG wire#powerrail
      I_Contact( "M_ZERO" )
      Not()
      wire#w1
      Contact( "M_0.5_SEC_2HZ" )
      wire#w2
      Coil( "SIGNAL_TWR_BLUE_LIGHT_Q" )
   END_RUNG
   RUNG wire#powerrail
      I_Contact( "M_ZERO" )
      Not()
   END_RUNG wire#w1
   RUNG wire#powerrail
      Contact( "M_ZERO" )
   END_RUNG wire#w2
   // the same network as SCL:
   "SIGNAL_TWR_BLUE_LIGHT_Q" := ((NOT (NOT "M_ZERO") OR NOT (NOT "M_ZERO")) AND "M_0.5_SEC_2HZ") OR "M_ZERO";
END_REGION

REGION Network 6: SIGNAL TOWER WHITE LIGHT OUTPUT / SIGNAL TOWER, BLUE LED
   // Blue Light
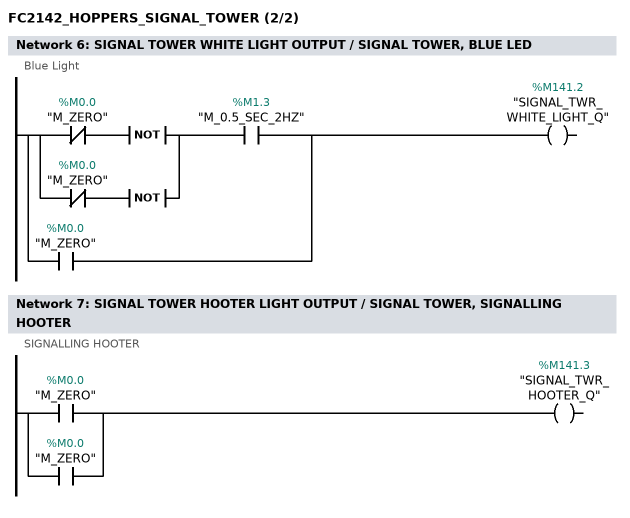
   RUNG wire#powerrail
      I_Contact( "M_ZERO" )
      Not()
      wire#w1
      Contact( "M_0.5_SEC_2HZ" )
      wire#w2
      Coil( "SIGNAL_TWR_WHITE_LIGHT_Q" )
   END_RUNG
   RUNG wire#powerrail
      I_Contact( "M_ZERO" )
      Not()
   END_RUNG wire#w1
   RUNG wire#powerrail
      Contact( "M_ZERO" )
   END_RUNG wire#w2
   // the same network as SCL:
   "SIGNAL_TWR_WHITE_LIGHT_Q" := ((NOT (NOT "M_ZERO") OR NOT (NOT "M_ZERO")) AND "M_0.5_SEC_2HZ") OR "M_ZERO";
END_REGION

REGION Network 7: SIGNAL TOWER HOOTER LIGHT OUTPUT / SIGNAL TOWER, SIGNALLING HOOTER
   // SIGNALLING HOOTER
   RUNG wire#powerrail
      Contact( "M_ZERO" )
      wire#w1
      Coil( "SIGNAL_TWR_HOOTER_Q" )
   END_RUNG
   RUNG wire#powerrail
      Contact( "M_ZERO" )
   END_RUNG wire#w1
   // the same network as SCL:
   "SIGNAL_TWR_HOOTER_Q" := "M_ZERO" OR "M_ZERO";
END_REGION
END_FUNCTION

FUNCTION "FC7200_HMI_HW_SW_DISABLE" : Void   // FC7200, LAD
{ S7_Optimized_Access := 'TRUE' }
VERSION : 0.1
// stored: AutoNumber false, IsIECCheckEnabled false, SetENOAutomatically false, UDAEnableTagReadback false
BEGIN

REGION Network 1: CALL FC7238 VARIABLES PLC CONNECTION
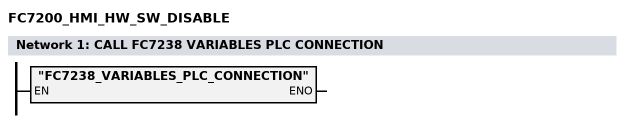
   RUNG wire#powerrail
      "FC7238_VARIABLES_PLC_CONNECTION"()
   END_RUNG
   // the same network as SCL:
   "FC7238_VARIABLES_PLC_CONNECTION"();
END_REGION
END_FUNCTION

FUNCTION "FC21000_POWDER_FEEDER_MAIN" : Void   // FC21000, LAD
TITLE = FC21000 POWDER FEEDER MAIN
{ S7_Optimized_Access := 'TRUE' }
VERSION : 0.1
// stored: AutoNumber false, IsIECCheckEnabled false, SetENOAutomatically false, UDAEnableTagReadback false
   VAR_TEMP
      ret_val_1 : Int;
      OPTIONS_OFF : Bool;
      OPTIONS_ON : Bool;
      POWDER_SWITCH_OPTION : Bool;
      MEDICOAT_OPTION : Bool;
   END_VAR
BEGIN

REGION Network 1: OPTIONS OFF
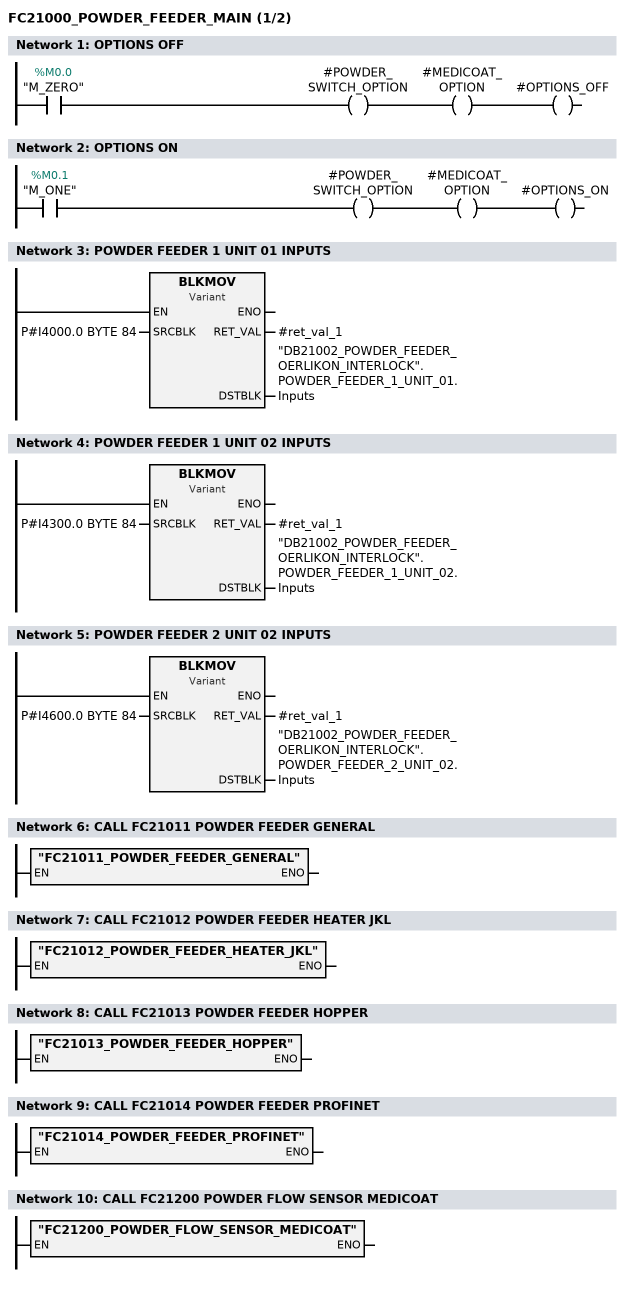
   RUNG wire#powerrail
      Contact( "M_ZERO" )
      Coil( #POWDER_SWITCH_OPTION )
      Coil( #MEDICOAT_OPTION )
      Coil( #OPTIONS_OFF )
   END_RUNG
   // the same network as SCL:
   #POWDER_SWITCH_OPTION := "M_ZERO";
   #MEDICOAT_OPTION := "M_ZERO";
   #OPTIONS_OFF := "M_ZERO";
END_REGION

REGION Network 2: OPTIONS ON
   RUNG wire#powerrail
      Contact( "M_ONE" )
      Coil( #POWDER_SWITCH_OPTION )
      Coil( #MEDICOAT_OPTION )
      Coil( #OPTIONS_ON )
   END_RUNG
   // the same network as SCL:
   #POWDER_SWITCH_OPTION := "M_ONE";
   #MEDICOAT_OPTION := "M_ONE";
   #OPTIONS_ON := "M_ONE";
END_REGION

REGION Network 3: POWDER FEEDER 1 UNIT 01 INPUTS
   RUNG wire#powerrail
      { S7_Templates := "blk_type := Variant" } BLKMOV(SRCBLK := P#I4000.0 BYTE 84, RET_VAL => #ret_val_1, DSTBLK => "DB21002_POWDER_FEEDER_OERLIKON_INTERLOCK".POWDER_FEEDER_1_UNIT_01.Inputs)
   END_RUNG
   // the same network as SCL:
   #ret_val_1 := BLKMOV(SRCBLK := P#I4000.0 BYTE 84,
                        DSTBLK => "DB21002_POWDER_FEEDER_OERLIKON_INTERLOCK".POWDER_FEEDER_1_UNIT_01.Inputs);
END_REGION

REGION Network 4: POWDER FEEDER 1 UNIT 02 INPUTS
   RUNG wire#powerrail
      { S7_Templates := "blk_type := Variant" } BLKMOV(SRCBLK := P#I4300.0 BYTE 84, RET_VAL => #ret_val_1, DSTBLK => "DB21002_POWDER_FEEDER_OERLIKON_INTERLOCK".POWDER_FEEDER_1_UNIT_02.Inputs)
   END_RUNG
   // the same network as SCL:
   #ret_val_1 := BLKMOV(SRCBLK := P#I4300.0 BYTE 84,
                        DSTBLK => "DB21002_POWDER_FEEDER_OERLIKON_INTERLOCK".POWDER_FEEDER_1_UNIT_02.Inputs);
END_REGION

REGION Network 5: POWDER FEEDER 2 UNIT 02 INPUTS
   RUNG wire#powerrail
      { S7_Templates := "blk_type := Variant" } BLKMOV(SRCBLK := P#I4600.0 BYTE 84, RET_VAL => #ret_val_1, DSTBLK => "DB21002_POWDER_FEEDER_OERLIKON_INTERLOCK".POWDER_FEEDER_2_UNIT_02.Inputs)
   END_RUNG
   // the same network as SCL:
   #ret_val_1 := BLKMOV(SRCBLK := P#I4600.0 BYTE 84,
                        DSTBLK => "DB21002_POWDER_FEEDER_OERLIKON_INTERLOCK".POWDER_FEEDER_2_UNIT_02.Inputs);
END_REGION

REGION Network 6: CALL FC21011 POWDER FEEDER GENERAL
   RUNG wire#powerrail
      "FC21011_POWDER_FEEDER_GENERAL"()
   END_RUNG
   // the same network as SCL:
   "FC21011_POWDER_FEEDER_GENERAL"();
END_REGION

REGION Network 7: CALL FC21012 POWDER FEEDER HEATER JKL
   RUNG wire#powerrail
      "FC21012_POWDER_FEEDER_HEATER_JKL"()
   END_RUNG
   // the same network as SCL:
   "FC21012_POWDER_FEEDER_HEATER_JKL"();
END_REGION

REGION Network 8: CALL FC21013 POWDER FEEDER HOPPER
   RUNG wire#powerrail
      "FC21013_POWDER_FEEDER_HOPPER"()
   END_RUNG
   // the same network as SCL:
   "FC21013_POWDER_FEEDER_HOPPER"();
END_REGION

REGION Network 9: CALL FC21014 POWDER FEEDER PROFINET
   RUNG wire#powerrail
      "FC21014_POWDER_FEEDER_PROFINET"()
   END_RUNG
   // the same network as SCL:
   "FC21014_POWDER_FEEDER_PROFINET"();
END_REGION

REGION Network 10: CALL FC21200 POWDER FLOW SENSOR MEDICOAT
   RUNG wire#powerrail
      "FC21200_POWDER_FLOW_SENSOR_MEDICOAT"()
   END_RUNG
   // the same network as SCL:
   "FC21200_POWDER_FLOW_SENSOR_MEDICOAT"();
END_REGION

REGION Network 11: POWDER FEEDER 1 UNIT 01 OUTPUTS
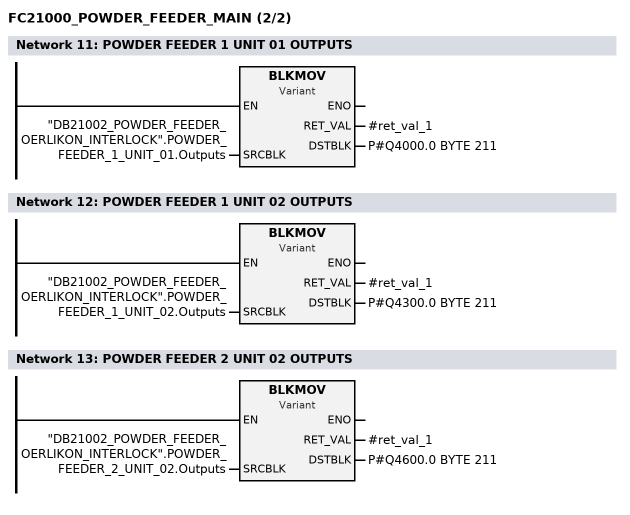
   RUNG wire#powerrail
      { S7_Templates := "blk_type := Variant" } BLKMOV(SRCBLK := "DB21002_POWDER_FEEDER_OERLIKON_INTERLOCK".POWDER_FEEDER_1_UNIT_01.Outputs, RET_VAL => #ret_val_1, DSTBLK => P#Q4000.0 BYTE 211)
   END_RUNG
   // the same network as SCL:
   #ret_val_1 := BLKMOV(SRCBLK := "DB21002_POWDER_FEEDER_OERLIKON_INTERLOCK".POWDER_FEEDER_1_UNIT_01.Outputs,
                        DSTBLK => P#Q4000.0 BYTE 211);
END_REGION

REGION Network 12: POWDER FEEDER 1 UNIT 02 OUTPUTS
   RUNG wire#powerrail
      { S7_Templates := "blk_type := Variant" } BLKMOV(SRCBLK := "DB21002_POWDER_FEEDER_OERLIKON_INTERLOCK".POWDER_FEEDER_1_UNIT_02.Outputs, RET_VAL => #ret_val_1, DSTBLK => P#Q4300.0 BYTE 211)
   END_RUNG
   // the same network as SCL:
   #ret_val_1 := BLKMOV(SRCBLK := "DB21002_POWDER_FEEDER_OERLIKON_INTERLOCK".POWDER_FEEDER_1_UNIT_02.Outputs,
                        DSTBLK => P#Q4300.0 BYTE 211);
END_REGION

REGION Network 13: POWDER FEEDER 2 UNIT 02 OUTPUTS
   RUNG wire#powerrail
      { S7_Templates := "blk_type := Variant" } BLKMOV(SRCBLK := "DB21002_POWDER_FEEDER_OERLIKON_INTERLOCK".POWDER_FEEDER_2_UNIT_02.Outputs, RET_VAL => #ret_val_1, DSTBLK => P#Q4600.0 BYTE 211)
   END_RUNG
   // the same network as SCL:
   #ret_val_1 := BLKMOV(SRCBLK := "DB21002_POWDER_FEEDER_OERLIKON_INTERLOCK".POWDER_FEEDER_2_UNIT_02.Outputs,
                        DSTBLK => P#Q4600.0 BYTE 211);
END_REGION
END_FUNCTION

FUNCTION "FC21011_POWDER_FEEDER_GENERAL" : Void   // FC21011, LAD
TITLE = FC21011 POWDER FEEDER GENERAL
{ S7_Optimized_Access := 'TRUE' }
VERSION : 0.1
// stored: AutoNumber false, IsIECCheckEnabled false, SetENOAutomatically false, UDAEnableTagReadback false
BEGIN

REGION Network 1: /////_UNIT_01_/////
END_REGION

REGION Network 2: CALL FB21011 POWDER FEEDER 1 GENERAL UNIT 01
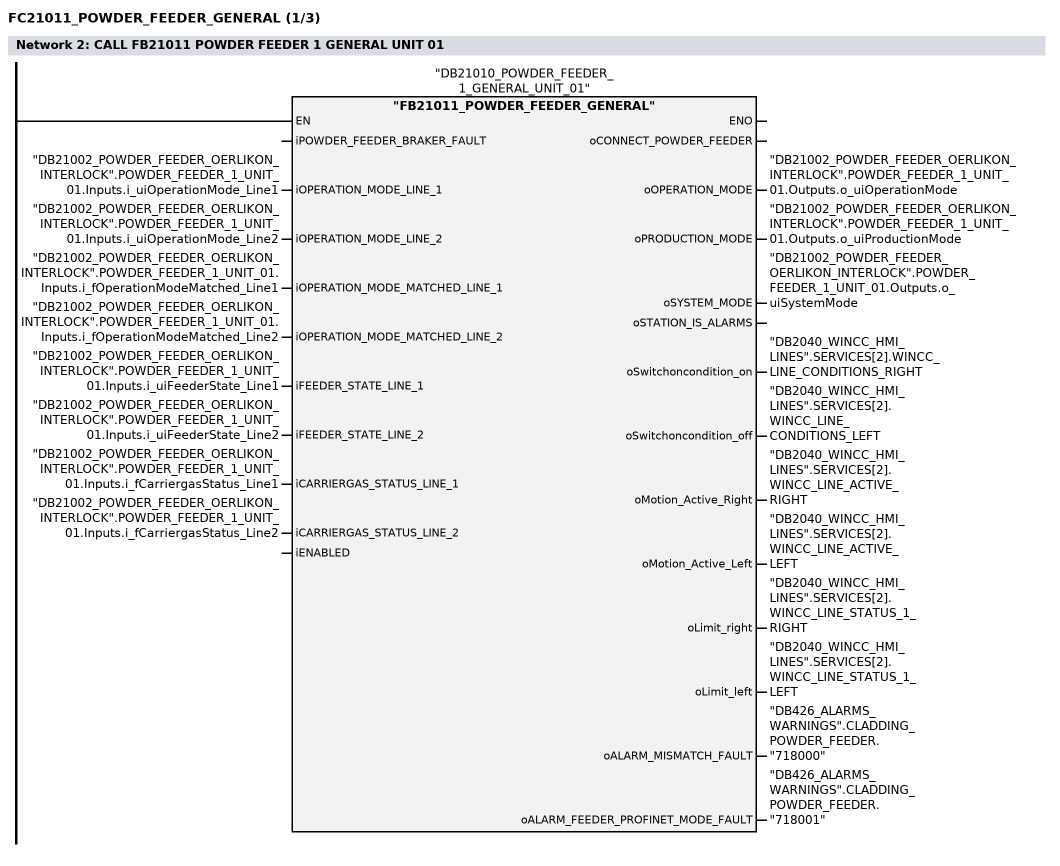
   RUNG wire#powerrail
      "DB21010_POWDER_FEEDER_1_GENERAL_UNIT_01"(iPOWDER_FEEDER_BRAKER_FAULT :=, iOPERATION_MODE_LINE_1 := "DB21002_POWDER_FEEDER_OERLIKON_INTERLOCK".POWDER_FEEDER_1_UNIT_01.Inputs.i_uiOperationMode_Line1, iOPERATION_MODE_LINE_2 := "DB21002_POWDER_FEEDER_OERLIKON_INTERLOCK".POWDER_FEEDER_1_UNIT_01.Inputs.i_uiOperationMode_Line2, iOPERATION_MODE_MATCHED_LINE_1 := "DB21002_POWDER_FEEDER_OERLIKON_INTERLOCK".POWDER_FEEDER_1_UNIT_01.Inputs.i_fOperationModeMatched_Line1, iOPERATION_MODE_MATCHED_LINE_2 := "DB21002_POWDER_FEEDER_OERLIKON_INTERLOCK".POWDER_FEEDER_1_UNIT_01.Inputs.i_fOperationModeMatched_Line2, iFEEDER_STATE_LINE_1 := "DB21002_POWDER_FEEDER_OERLIKON_INTERLOCK".POWDER_FEEDER_1_UNIT_01.Inputs.i_uiFeederState_Line1, iFEEDER_STATE_LINE_2 := "DB21002_POWDER_FEEDER_OERLIKON_INTERLOCK".POWDER_FEEDER_1_UNIT_01.Inputs.i_uiFeederState_Line2, iCARRIERGAS_STATUS_LINE_1 := "DB21002_POWDER_FEEDER_OERLIKON_INTERLOCK".POWDER_FEEDER_1_UNIT_01.Inputs.i_fCarriergasStatus_Line1, iCARRIERGAS_STATUS_LINE_2 := "DB21002_POWDER_FEEDER_OERLIKON_INTERLOCK".POWDER_FEEDER_1_UNIT_01.Inputs.i_fCarriergasStatus_Line2, iENABLED :=, oCONNECT_POWDER_FEEDER =>, oOPERATION_MODE => "DB21002_POWDER_FEEDER_OERLIKON_INTERLOCK".POWDER_FEEDER_1_UNIT_01.Outputs.o_uiOperationMode, oPRODUCTION_MODE => "DB21002_POWDER_FEEDER_OERLIKON_INTERLOCK".POWDER_FEEDER_1_UNIT_01.Outputs.o_uiProductionMode, oSYSTEM_MODE => "DB21002_POWDER_FEEDER_OERLIKON_INTERLOCK".POWDER_FEEDER_1_UNIT_01.Outputs.o_uiSystemMode, oSTATION_IS_ALARMS =>, oSwitchoncondition_on => "DB2040_WINCC_HMI_LINES".SERVICES[2].WINCC_LINE_CONDITIONS_RIGHT, oSwitchoncondition_off => "DB2040_WINCC_HMI_LINES".SERVICES[2].WINCC_LINE_CONDITIONS_LEFT, oMotion_Active_Right => "DB2040_WINCC_HMI_LINES".SERVICES[2].WINCC_LINE_ACTIVE_RIGHT, oMotion_Active_Left => "DB2040_WINCC_HMI_LINES".SERVICES[2].WINCC_LINE_ACTIVE_LEFT, oLimit_right => "DB2040_WINCC_HMI_LINES".SERVICES[2].WINCC_LINE_STATUS_1_RIGHT, oLimit_left => "DB2040_WINCC_HMI_LINES".SERVICES[2].WINCC_LINE_STATUS_1_LEFT, oALARM_MISMATCH_FAULT => "DB426_ALARMS_WARNINGS".CLADDING_POWDER_FEEDER."718000", oALARM_FEEDER_PROFINET_MODE_FAULT => "DB426_ALARMS_WARNINGS".CLADDING_POWDER_FEEDER."718001")
   END_RUNG
   // the same network as SCL:
   "DB21010_POWDER_FEEDER_1_GENERAL_UNIT_01"(iOPERATION_MODE_LINE_1 := "DB21002_POWDER_FEEDER_OERLIKON_INTERLOCK".POWDER_FEEDER_1_UNIT_01.Inputs.i_uiOperationMode_Line1,   // "FB21011_POWDER_FEEDER_GENERAL"
                           iOPERATION_MODE_LINE_2 := "DB21002_POWDER_FEEDER_OERLIKON_INTERLOCK".POWDER_FEEDER_1_UNIT_01.Inputs.i_uiOperationMode_Line2,
                           iOPERATION_MODE_MATCHED_LINE_1 := "DB21002_POWDER_FEEDER_OERLIKON_INTERLOCK".POWDER_FEEDER_1_UNIT_01.Inputs.i_fOperationModeMatched_Line1,
                           iOPERATION_MODE_MATCHED_LINE_2 := "DB21002_POWDER_FEEDER_OERLIKON_INTERLOCK".POWDER_FEEDER_1_UNIT_01.Inputs.i_fOperationModeMatched_Line2,
                           iFEEDER_STATE_LINE_1 := "DB21002_POWDER_FEEDER_OERLIKON_INTERLOCK".POWDER_FEEDER_1_UNIT_01.Inputs.i_uiFeederState_Line1,
                           iFEEDER_STATE_LINE_2 := "DB21002_POWDER_FEEDER_OERLIKON_INTERLOCK".POWDER_FEEDER_1_UNIT_01.Inputs.i_uiFeederState_Line2,
                           iCARRIERGAS_STATUS_LINE_1 := "DB21002_POWDER_FEEDER_OERLIKON_INTERLOCK".POWDER_FEEDER_1_UNIT_01.Inputs.i_fCarriergasStatus_Line1,
                           iCARRIERGAS_STATUS_LINE_2 := "DB21002_POWDER_FEEDER_OERLIKON_INTERLOCK".POWDER_FEEDER_1_UNIT_01.Inputs.i_fCarriergasStatus_Line2,
                           oOPERATION_MODE => "DB21002_POWDER_FEEDER_OERLIKON_INTERLOCK".POWDER_FEEDER_1_UNIT_01.Outputs.o_uiOperationMode,
                           oPRODUCTION_MODE => "DB21002_POWDER_FEEDER_OERLIKON_INTERLOCK".POWDER_FEEDER_1_UNIT_01.Outputs.o_uiProductionMode,
                           oSYSTEM_MODE => "DB21002_POWDER_FEEDER_OERLIKON_INTERLOCK".POWDER_FEEDER_1_UNIT_01.Outputs.o_uiSystemMode,
                           oSwitchoncondition_on => "DB2040_WINCC_HMI_LINES".SERVICES[2].WINCC_LINE_CONDITIONS_RIGHT,
                           oSwitchoncondition_off => "DB2040_WINCC_HMI_LINES".SERVICES[2].WINCC_LINE_CONDITIONS_LEFT,
                           oMotion_Active_Right => "DB2040_WINCC_HMI_LINES".SERVICES[2].WINCC_LINE_ACTIVE_RIGHT,
                           oMotion_Active_Left => "DB2040_WINCC_HMI_LINES".SERVICES[2].WINCC_LINE_ACTIVE_LEFT,
                           oLimit_right => "DB2040_WINCC_HMI_LINES".SERVICES[2].WINCC_LINE_STATUS_1_RIGHT,
                           oLimit_left => "DB2040_WINCC_HMI_LINES".SERVICES[2].WINCC_LINE_STATUS_1_LEFT,
                           oALARM_MISMATCH_FAULT => "DB426_ALARMS_WARNINGS".CLADDING_POWDER_FEEDER."718000",
                           oALARM_FEEDER_PROFINET_MODE_FAULT => "DB426_ALARMS_WARNINGS".CLADDING_POWDER_FEEDER."718001");
END_REGION

REGION Network 3: /////_UNIT_02_/////
END_REGION

REGION Network 4: CALL FB21011 POWDER FEEDER 1 GENERAL UNIT 02
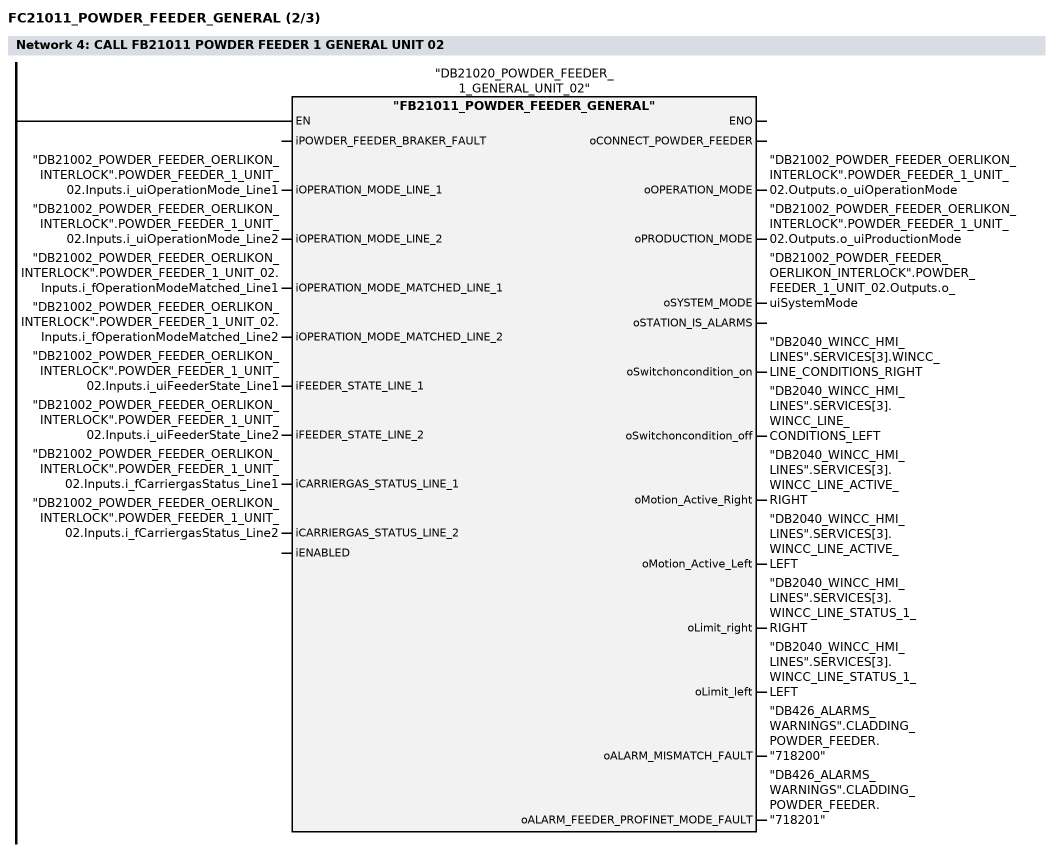
   RUNG wire#powerrail
      "DB21020_POWDER_FEEDER_1_GENERAL_UNIT_02"(iPOWDER_FEEDER_BRAKER_FAULT :=, iOPERATION_MODE_LINE_1 := "DB21002_POWDER_FEEDER_OERLIKON_INTERLOCK".POWDER_FEEDER_1_UNIT_02.Inputs.i_uiOperationMode_Line1, iOPERATION_MODE_LINE_2 := "DB21002_POWDER_FEEDER_OERLIKON_INTERLOCK".POWDER_FEEDER_1_UNIT_02.Inputs.i_uiOperationMode_Line2, iOPERATION_MODE_MATCHED_LINE_1 := "DB21002_POWDER_FEEDER_OERLIKON_INTERLOCK".POWDER_FEEDER_1_UNIT_02.Inputs.i_fOperationModeMatched_Line1, iOPERATION_MODE_MATCHED_LINE_2 := "DB21002_POWDER_FEEDER_OERLIKON_INTERLOCK".POWDER_FEEDER_1_UNIT_02.Inputs.i_fOperationModeMatched_Line2, iFEEDER_STATE_LINE_1 := "DB21002_POWDER_FEEDER_OERLIKON_INTERLOCK".POWDER_FEEDER_1_UNIT_02.Inputs.i_uiFeederState_Line1, iFEEDER_STATE_LINE_2 := "DB21002_POWDER_FEEDER_OERLIKON_INTERLOCK".POWDER_FEEDER_1_UNIT_02.Inputs.i_uiFeederState_Line2, iCARRIERGAS_STATUS_LINE_1 := "DB21002_POWDER_FEEDER_OERLIKON_INTERLOCK".POWDER_FEEDER_1_UNIT_02.Inputs.i_fCarriergasStatus_Line1, iCARRIERGAS_STATUS_LINE_2 := "DB21002_POWDER_FEEDER_OERLIKON_INTERLOCK".POWDER_FEEDER_1_UNIT_02.Inputs.i_fCarriergasStatus_Line2, iENABLED :=, oCONNECT_POWDER_FEEDER =>, oOPERATION_MODE => "DB21002_POWDER_FEEDER_OERLIKON_INTERLOCK".POWDER_FEEDER_1_UNIT_02.Outputs.o_uiOperationMode, oPRODUCTION_MODE => "DB21002_POWDER_FEEDER_OERLIKON_INTERLOCK".POWDER_FEEDER_1_UNIT_02.Outputs.o_uiProductionMode, oSYSTEM_MODE => "DB21002_POWDER_FEEDER_OERLIKON_INTERLOCK".POWDER_FEEDER_1_UNIT_02.Outputs.o_uiSystemMode, oSTATION_IS_ALARMS =>, oSwitchoncondition_on => "DB2040_WINCC_HMI_LINES".SERVICES[3].WINCC_LINE_CONDITIONS_RIGHT, oSwitchoncondition_off => "DB2040_WINCC_HMI_LINES".SERVICES[3].WINCC_LINE_CONDITIONS_LEFT, oMotion_Active_Right => "DB2040_WINCC_HMI_LINES".SERVICES[3].WINCC_LINE_ACTIVE_RIGHT, oMotion_Active_Left => "DB2040_WINCC_HMI_LINES".SERVICES[3].WINCC_LINE_ACTIVE_LEFT, oLimit_right => "DB2040_WINCC_HMI_LINES".SERVICES[3].WINCC_LINE_STATUS_1_RIGHT, oLimit_left => "DB2040_WINCC_HMI_LINES".SERVICES[3].WINCC_LINE_STATUS_1_LEFT, oALARM_MISMATCH_FAULT => "DB426_ALARMS_WARNINGS".CLADDING_POWDER_FEEDER."718200", oALARM_FEEDER_PROFINET_MODE_FAULT => "DB426_ALARMS_WARNINGS".CLADDING_POWDER_FEEDER."718201")
   END_RUNG
   // the same network as SCL:
   "DB21020_POWDER_FEEDER_1_GENERAL_UNIT_02"(iOPERATION_MODE_LINE_1 := "DB21002_POWDER_FEEDER_OERLIKON_INTERLOCK".POWDER_FEEDER_1_UNIT_02.Inputs.i_uiOperationMode_Line1,   // "FB21011_POWDER_FEEDER_GENERAL"
                           iOPERATION_MODE_LINE_2 := "DB21002_POWDER_FEEDER_OERLIKON_INTERLOCK".POWDER_FEEDER_1_UNIT_02.Inputs.i_uiOperationMode_Line2,
                           iOPERATION_MODE_MATCHED_LINE_1 := "DB21002_POWDER_FEEDER_OERLIKON_INTERLOCK".POWDER_FEEDER_1_UNIT_02.Inputs.i_fOperationModeMatched_Line1,
                           iOPERATION_MODE_MATCHED_LINE_2 := "DB21002_POWDER_FEEDER_OERLIKON_INTERLOCK".POWDER_FEEDER_1_UNIT_02.Inputs.i_fOperationModeMatched_Line2,
                           iFEEDER_STATE_LINE_1 := "DB21002_POWDER_FEEDER_OERLIKON_INTERLOCK".POWDER_FEEDER_1_UNIT_02.Inputs.i_uiFeederState_Line1,
                           iFEEDER_STATE_LINE_2 := "DB21002_POWDER_FEEDER_OERLIKON_INTERLOCK".POWDER_FEEDER_1_UNIT_02.Inputs.i_uiFeederState_Line2,
                           iCARRIERGAS_STATUS_LINE_1 := "DB21002_POWDER_FEEDER_OERLIKON_INTERLOCK".POWDER_FEEDER_1_UNIT_02.Inputs.i_fCarriergasStatus_Line1,
                           iCARRIERGAS_STATUS_LINE_2 := "DB21002_POWDER_FEEDER_OERLIKON_INTERLOCK".POWDER_FEEDER_1_UNIT_02.Inputs.i_fCarriergasStatus_Line2,
                           oOPERATION_MODE => "DB21002_POWDER_FEEDER_OERLIKON_INTERLOCK".POWDER_FEEDER_1_UNIT_02.Outputs.o_uiOperationMode,
                           oPRODUCTION_MODE => "DB21002_POWDER_FEEDER_OERLIKON_INTERLOCK".POWDER_FEEDER_1_UNIT_02.Outputs.o_uiProductionMode,
                           oSYSTEM_MODE => "DB21002_POWDER_FEEDER_OERLIKON_INTERLOCK".POWDER_FEEDER_1_UNIT_02.Outputs.o_uiSystemMode,
                           oSwitchoncondition_on => "DB2040_WINCC_HMI_LINES".SERVICES[3].WINCC_LINE_CONDITIONS_RIGHT,
                           oSwitchoncondition_off => "DB2040_WINCC_HMI_LINES".SERVICES[3].WINCC_LINE_CONDITIONS_LEFT,
                           oMotion_Active_Right => "DB2040_WINCC_HMI_LINES".SERVICES[3].WINCC_LINE_ACTIVE_RIGHT,
                           oMotion_Active_Left => "DB2040_WINCC_HMI_LINES".SERVICES[3].WINCC_LINE_ACTIVE_LEFT,
                           oLimit_right => "DB2040_WINCC_HMI_LINES".SERVICES[3].WINCC_LINE_STATUS_1_RIGHT,
                           oLimit_left => "DB2040_WINCC_HMI_LINES".SERVICES[3].WINCC_LINE_STATUS_1_LEFT,
                           oALARM_MISMATCH_FAULT => "DB426_ALARMS_WARNINGS".CLADDING_POWDER_FEEDER."718200",
                           oALARM_FEEDER_PROFINET_MODE_FAULT => "DB426_ALARMS_WARNINGS".CLADDING_POWDER_FEEDER."718201");
END_REGION

REGION Network 5: CALL FB21011 POWDER FEEDER 2 GENERAL UNIT 02
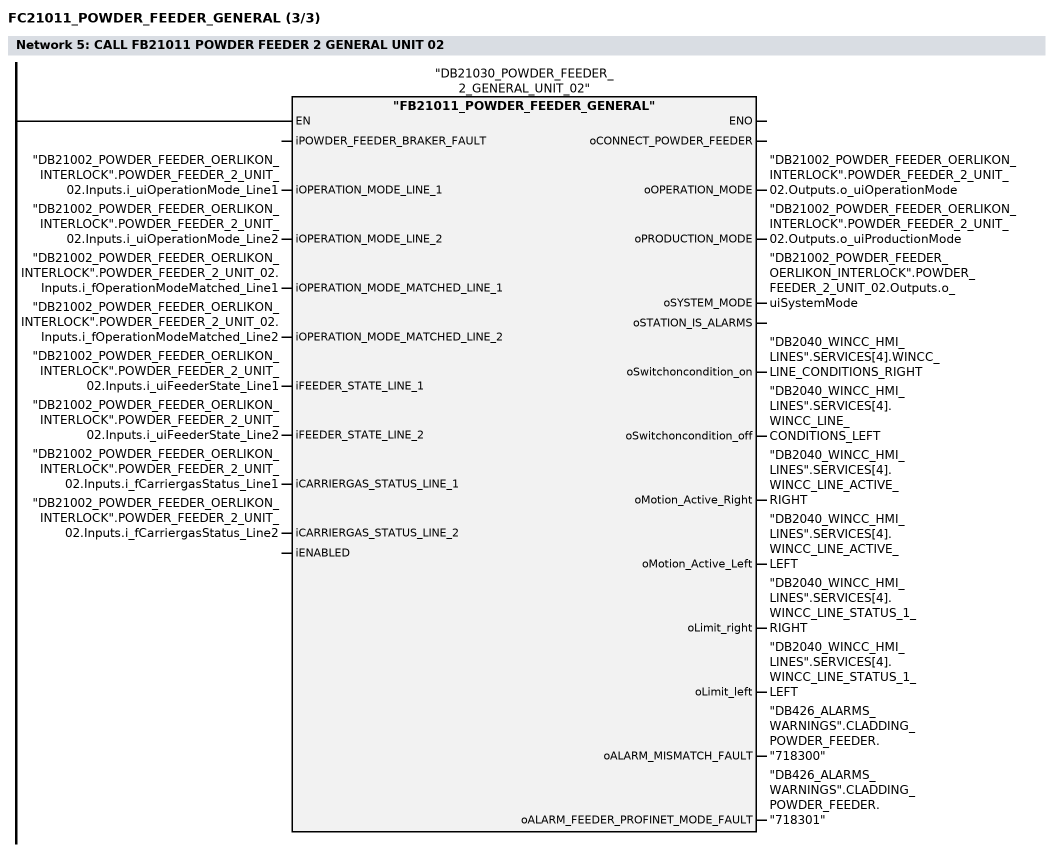
   RUNG wire#powerrail
      "DB21030_POWDER_FEEDER_2_GENERAL_UNIT_02"(iPOWDER_FEEDER_BRAKER_FAULT :=, iOPERATION_MODE_LINE_1 := "DB21002_POWDER_FEEDER_OERLIKON_INTERLOCK".POWDER_FEEDER_2_UNIT_02.Inputs.i_uiOperationMode_Line1, iOPERATION_MODE_LINE_2 := "DB21002_POWDER_FEEDER_OERLIKON_INTERLOCK".POWDER_FEEDER_2_UNIT_02.Inputs.i_uiOperationMode_Line2, iOPERATION_MODE_MATCHED_LINE_1 := "DB21002_POWDER_FEEDER_OERLIKON_INTERLOCK".POWDER_FEEDER_2_UNIT_02.Inputs.i_fOperationModeMatched_Line1, iOPERATION_MODE_MATCHED_LINE_2 := "DB21002_POWDER_FEEDER_OERLIKON_INTERLOCK".POWDER_FEEDER_2_UNIT_02.Inputs.i_fOperationModeMatched_Line2, iFEEDER_STATE_LINE_1 := "DB21002_POWDER_FEEDER_OERLIKON_INTERLOCK".POWDER_FEEDER_2_UNIT_02.Inputs.i_uiFeederState_Line1, iFEEDER_STATE_LINE_2 := "DB21002_POWDER_FEEDER_OERLIKON_INTERLOCK".POWDER_FEEDER_2_UNIT_02.Inputs.i_uiFeederState_Line2, iCARRIERGAS_STATUS_LINE_1 := "DB21002_POWDER_FEEDER_OERLIKON_INTERLOCK".POWDER_FEEDER_2_UNIT_02.Inputs.i_fCarriergasStatus_Line1, iCARRIERGAS_STATUS_LINE_2 := "DB21002_POWDER_FEEDER_OERLIKON_INTERLOCK".POWDER_FEEDER_2_UNIT_02.Inputs.i_fCarriergasStatus_Line2, iENABLED :=, oCONNECT_POWDER_FEEDER =>, oOPERATION_MODE => "DB21002_POWDER_FEEDER_OERLIKON_INTERLOCK".POWDER_FEEDER_2_UNIT_02.Outputs.o_uiOperationMode, oPRODUCTION_MODE => "DB21002_POWDER_FEEDER_OERLIKON_INTERLOCK".POWDER_FEEDER_2_UNIT_02.Outputs.o_uiProductionMode, oSYSTEM_MODE => "DB21002_POWDER_FEEDER_OERLIKON_INTERLOCK".POWDER_FEEDER_2_UNIT_02.Outputs.o_uiSystemMode, oSTATION_IS_ALARMS =>, oSwitchoncondition_on => "DB2040_WINCC_HMI_LINES".SERVICES[4].WINCC_LINE_CONDITIONS_RIGHT, oSwitchoncondition_off => "DB2040_WINCC_HMI_LINES".SERVICES[4].WINCC_LINE_CONDITIONS_LEFT, oMotion_Active_Right => "DB2040_WINCC_HMI_LINES".SERVICES[4].WINCC_LINE_ACTIVE_RIGHT, oMotion_Active_Left => "DB2040_WINCC_HMI_LINES".SERVICES[4].WINCC_LINE_ACTIVE_LEFT, oLimit_right => "DB2040_WINCC_HMI_LINES".SERVICES[4].WINCC_LINE_STATUS_1_RIGHT, oLimit_left => "DB2040_WINCC_HMI_LINES".SERVICES[4].WINCC_LINE_STATUS_1_LEFT, oALARM_MISMATCH_FAULT => "DB426_ALARMS_WARNINGS".CLADDING_POWDER_FEEDER."718300", oALARM_FEEDER_PROFINET_MODE_FAULT => "DB426_ALARMS_WARNINGS".CLADDING_POWDER_FEEDER."718301")
   END_RUNG
   // the same network as SCL:
   "DB21030_POWDER_FEEDER_2_GENERAL_UNIT_02"(iOPERATION_MODE_LINE_1 := "DB21002_POWDER_FEEDER_OERLIKON_INTERLOCK".POWDER_FEEDER_2_UNIT_02.Inputs.i_uiOperationMode_Line1,   // "FB21011_POWDER_FEEDER_GENERAL"
                           iOPERATION_MODE_LINE_2 := "DB21002_POWDER_FEEDER_OERLIKON_INTERLOCK".POWDER_FEEDER_2_UNIT_02.Inputs.i_uiOperationMode_Line2,
                           iOPERATION_MODE_MATCHED_LINE_1 := "DB21002_POWDER_FEEDER_OERLIKON_INTERLOCK".POWDER_FEEDER_2_UNIT_02.Inputs.i_fOperationModeMatched_Line1,
                           iOPERATION_MODE_MATCHED_LINE_2 := "DB21002_POWDER_FEEDER_OERLIKON_INTERLOCK".POWDER_FEEDER_2_UNIT_02.Inputs.i_fOperationModeMatched_Line2,
                           iFEEDER_STATE_LINE_1 := "DB21002_POWDER_FEEDER_OERLIKON_INTERLOCK".POWDER_FEEDER_2_UNIT_02.Inputs.i_uiFeederState_Line1,
                           iFEEDER_STATE_LINE_2 := "DB21002_POWDER_FEEDER_OERLIKON_INTERLOCK".POWDER_FEEDER_2_UNIT_02.Inputs.i_uiFeederState_Line2,
                           iCARRIERGAS_STATUS_LINE_1 := "DB21002_POWDER_FEEDER_OERLIKON_INTERLOCK".POWDER_FEEDER_2_UNIT_02.Inputs.i_fCarriergasStatus_Line1,
                           iCARRIERGAS_STATUS_LINE_2 := "DB21002_POWDER_FEEDER_OERLIKON_INTERLOCK".POWDER_FEEDER_2_UNIT_02.Inputs.i_fCarriergasStatus_Line2,
                           oOPERATION_MODE => "DB21002_POWDER_FEEDER_OERLIKON_INTERLOCK".POWDER_FEEDER_2_UNIT_02.Outputs.o_uiOperationMode,
                           oPRODUCTION_MODE => "DB21002_POWDER_FEEDER_OERLIKON_INTERLOCK".POWDER_FEEDER_2_UNIT_02.Outputs.o_uiProductionMode,
                           oSYSTEM_MODE => "DB21002_POWDER_FEEDER_OERLIKON_INTERLOCK".POWDER_FEEDER_2_UNIT_02.Outputs.o_uiSystemMode,
                           oSwitchoncondition_on => "DB2040_WINCC_HMI_LINES".SERVICES[4].WINCC_LINE_CONDITIONS_RIGHT,
                           oSwitchoncondition_off => "DB2040_WINCC_HMI_LINES".SERVICES[4].WINCC_LINE_CONDITIONS_LEFT,
                           oMotion_Active_Right => "DB2040_WINCC_HMI_LINES".SERVICES[4].WINCC_LINE_ACTIVE_RIGHT,
                           oMotion_Active_Left => "DB2040_WINCC_HMI_LINES".SERVICES[4].WINCC_LINE_ACTIVE_LEFT,
                           oLimit_right => "DB2040_WINCC_HMI_LINES".SERVICES[4].WINCC_LINE_STATUS_1_RIGHT,
                           oLimit_left => "DB2040_WINCC_HMI_LINES".SERVICES[4].WINCC_LINE_STATUS_1_LEFT,
                           oALARM_MISMATCH_FAULT => "DB426_ALARMS_WARNINGS".CLADDING_POWDER_FEEDER."718300",
                           oALARM_FEEDER_PROFINET_MODE_FAULT => "DB426_ALARMS_WARNINGS".CLADDING_POWDER_FEEDER."718301");
END_REGION
END_FUNCTION

FUNCTION_BLOCK "FB21011_POWDER_FEEDER_GENERAL"   // FB21011, LAD
TITLE = FB21011 POWDER FEEDER GENERAL
{ S7_Optimized_Access := 'TRUE' }
VERSION : 0.1
// stored: AutoNumber false, IsIECCheckEnabled false, IsRetainMemResEnabled false, MemoryReserve 100, SetENOAutomatically false, UDAEnableTagReadback false
   VAR_INPUT
      iPOWDER_FEEDER_BRAKER_FAULT : Bool;
      iOPERATION_MODE_LINE_1 : Word;
      iOPERATION_MODE_LINE_2 : Word;
      iOPERATION_MODE_MATCHED_LINE_1 : Bool;
      iOPERATION_MODE_MATCHED_LINE_2 : Bool;
      iFEEDER_STATE_LINE_1 : Word;
      iFEEDER_STATE_LINE_2 : Word;
      iCARRIERGAS_STATUS_LINE_1 : Bool;
      iCARRIERGAS_STATUS_LINE_2 : Bool;
      iENABLED : Bool;
   END_VAR
   VAR_OUTPUT
      oCONNECT_POWDER_FEEDER : Bool;
      oOPERATION_MODE : Word;
      oPRODUCTION_MODE : Word;
      oSYSTEM_MODE : Word;
      oSTATION_IS_ALARMS : Bool;
      oSwitchoncondition_on : Bool;
      oSwitchoncondition_off : Bool;
      oMotion_Active_Right : Bool;
      oMotion_Active_Left : Bool;
      oLimit_right : Bool;
      oLimit_left : Bool;
      oALARM_MISMATCH_FAULT : Bool;
      oALARM_FEEDER_PROFINET_MODE_FAULT : Bool;
   END_VAR
   VAR
      DATA : "POWDER FEEDER GENERAL";
      INPUT_SETTINGS : Struct
         UNIT_NUMBER : Int;
         FEEDER_NUMBER : Int;
      END_STRUCT;
   END_VAR
   VAR_TEMP
      OPTIONS_OFF : Bool;
      OPTIONS_ON : Bool;
      HOPPER_1 : Bool;
      HOPPER_2 : Bool;
      DB_NUMBER : DInt;
   END_VAR
   VAR_TEMP   // added for the SCL form of the ladder/FBD networks
      _w1 : Bool;
   END_VAR
BEGIN

NETWORK
TITLE = READ INSTANCE DB NUMBER
      L     DINO;
      +     10#800000;
      T     #DB_NUMBER;

REGION Network 2: OPTIONS OFF / Options Off
